	            #iqUDT_ConveyorInterface.VFDatSpeed := #sx_SpeedSetpointReached AND
	            #sx_AixAvailableControler AND
	            #si_ActualSpeed <> 0 AND
	            NOT #sx_SpeedFeedbackError;             // Copy setpoint speed reached state from static to the output conveyor interface structure

	            #iqUDT_ConveyorInterface.InternalWarningVFD := #sUDT_HMIStatus.PNSlaveWarning;                                                       // Set the internal warning bit if any warning is active

	            #iqUDT_ConveyorInterface.InternalErrorVFD := #sx_ErrorCMotor;                   // Set the internal error bit if any fault is active

	            #iqUDT_ConveyorInterface.ActualSpeed := ABS(#si_ActualSpeed);                   // Copy the calculated value to the output

	            #iqUDT_ConveyorInterface.ConfigurationError := #sx_ConfigurationError;          // Copy the calculated value to the output

	        END_IF;


	    END_REGION

	    REGION 10.2 - Move error status TO HMI Status

	        // Copy error status to output
	        #qUDT_HMIStatus := #sUDT_HMIStatus;

	    END_REGION

	END_REGION

	REGION 11 - Statistic

	    REGION 11.1 - General
	        // Statement section REGION
	        #sx_GeneralStatisticsReset := #iqUDT_ConveyorInterface.ResetStatistics;
	    END_REGION

	    // Create trigger on error and create statistics for profinet slave not online
	    #sR_TRIG_PNSlaveNotOnline(CLK := #sUDT_HMIStatus.PNSlaveNotOnline);                 // Detect the rising edge of the error

	    IF #sx_GeneralStatisticsReset OR #sUDT_HMIStatus.PNSlaveNotOnline
	    THEN

	        "FC_Statistics"(ix_Reset := #sx_GeneralStatisticsReset,
	                        ix_Activate := #sUDT_HMIStatus.PNSlaveNotOnline,
	                        ix_RTrigActivate := #sR_TRIG_PNSlaveNotOnline.Q,
	                        iqUDT_Statistics := #iqUDT_MCOStatistics.PNSlaveNotOnline);

	        #iqUDT_MCOStatistics.PNSlaveNotOnline := #iqUDT_MCOStatistics.PNSlaveNotOnline;
	    END_IF;

	    // Create trigger on error and create statistics for profinet slave error
	    #sR_TRIG_PNSlaveError(CLK := #sUDT_HMIStatus.PNSlaveError);                                                                          // Detect the rising edge of the error

	    IF #sx_GeneralStatisticsReset OR #sUDT_HMIStatus.PNSlaveError
	    THEN

	        "FC_Statistics"(ix_Reset := #sx_GeneralStatisticsReset,
	                        ix_Activate := #sUDT_HMIStatus.PNSlaveError,
	                        ix_RTrigActivate := #sR_TRIG_PNSlaveError.Q,
	                        iqUDT_Statistics := #iqUDT_MCOStatistics.PNSlaveError);

	        #iqUDT_MCOStatistics.PNSlaveError := #iqUDT_MCOStatistics.PNSlaveError;
	    END_IF;


	    // Create trigger on error and create statistics for MCO communication error
	    #sR_TRIG_CommunicationErrorMCO(CLK := #qUDT_HMIStatus.CommunicationErrorVFD);            // Detect the rising edge of the error

	    IF #sx_GeneralStatisticsReset OR #qUDT_HMIStatus.CommunicationErrorVFD
	    THEN

	        "FC_Statistics"(ix_Reset := #sx_GeneralStatisticsReset,
	                        ix_Activate := #qUDT_HMIStatus.CommunicationErrorVFD,
	                        ix_RTrigActivate := #sR_TRIG_CommunicationErrorMCO.Q,
	                        iqUDT_Statistics := #iqUDT_MCOStatistics.CommunicationErrorMovikit);

	    END_IF;

	    REGION 11.1 - Motor

	        // Create trigger on error and create statistics for internal MCO Error
	        #sR_TRIG_MCOInternalError(CLK := #sUDT_HMIStatus.InternalError);         // Detect the rising edge of the error

	        IF #iqUDT_ConveyorInterface.ResetStatistics OR #sUDT_HMIStatus.InternalError
	        THEN

	            "FC_Statistics"(ix_Reset := #iqUDT_ConveyorInterface.ResetStatistics,
	                            ix_Activate := #sUDT_HMIStatus.InternalError,
	                            ix_RTrigActivate := #sR_TRIG_MCOInternalError.Q,
	                            iqUDT_Statistics := #iqUDT_MCOStatistics.VFDInternalError);

	        END_IF;

	        // Create trigger on running signal and create statistics for running status
	        #sR_TRIG_Running(CLK := #iqUDT_ConveyorInterface.VFDRunning);                           // Detect the rising edge of the signal

	        IF #iqUDT_ConveyorInterface.ResetStatistics OR #iqUDT_ConveyorInterface.VFDRunning
	        THEN

	            "FC_Statistics"(ix_Reset := #iqUDT_ConveyorInterface.ResetStatistics,
	                            ix_Activate := #iqUDT_ConveyorInterface.VFDRunning,
	                            ix_RTrigActivate := #sR_TRIG_Running.Q,
	                            iqUDT_Statistics := #iqUDT_MCOStatistics.Running);
	        END_IF;


	    END_REGION
	    REGION 12 Status bit allocation
	        "FC_BitAllocation"(ix_Bit0 := #qUDT_HMIStatus.SpeedFeedbackError,
	                           ix_Bit1 := #qUDT_HMIStatus.InternalWarning,
	                           ix_Bit2 := #qUDT_HMIStatus.InternalError,
	                           ix_Bit3 := #qUDT_HMIStatus.CommunicationErrorVFD,
	                           ix_Bit4 := #qUDT_HMIStatus.PNSlaveNotOnline,
	                           ix_Bit5 := #qUDT_HMIStatus.PNSlaveError,
	                           ix_Bit6 := #qUDT_HMIStatus.PNSlaveWarning,
	                           ix_Bit7 := FALSE,
	                           ix_Bit8 := FALSE,
	                           ix_Bit9 := FALSE,
	                           ix_Bit10 := FALSE,
	                           ix_Bit11 := FALSE,
	                           ix_Bit12 := FALSE,
	                           ix_Bit13 := FALSE,
	                           ix_Bit14 := FALSE,
	                           ix_Bit15 := FALSE,
	                           ix_Bit16 := FALSE,
	                           ix_Bit17 := FALSE,
	                           ix_Bit18 := FALSE,
	                           ix_Bit19 := FALSE,
	                           ix_Bit20 := FALSE,
	                           ix_Bit21 := FALSE,
	                           ix_Bit22 := FALSE,
	                           ix_Bit23 := FALSE,
	                           ix_Bit24 := FALSE,
	                           ix_Bit25 := FALSE,
	                           ix_Bit26 := FALSE,
	                           ix_Bit27 := FALSE,
	                           ix_Bit28 := FALSE,
	                           ix_Bit29 := FALSE,
	                           ix_Bit30 := FALSE,
	                           ix_Bit31 := FALSE,
	                           qdw_Dword => #qUDT_HMIStatus.ControllerStatus);
	    END_REGION
	END_REGION
END_FUNCTION_BLOCK

FUNCTION_BLOCK "FB_GateSection"
{ S7_Optimized_Access := 'TRUE' }
VERSION : 0.1
// ATTRIBUTES
// AUTO_NUMBER = True
// BLOCK_NUMBER = 213
// END_ATTRIBUTES
   VAR_INPUT
      ix_GateOpen { ExternalAccessible := 'False'; ExternalVisible := 'False'; ExternalWritable := 'False'} : Bool;   // When TRUE gate is open, when FALSE gate is close
      ix_OperatorButton { ExternalAccessible := 'False'; ExternalVisible := 'False'; ExternalWritable := 'False'} : Bool;   // When TRUE then operator button is pressed
      iudi_TimeOnDelay { ExternalAccessible := 'False'; ExternalVisible := 'False'; ExternalWritable := 'False'} : UDInt;   // Time on delay to enable the horn when the gate is closed
   END_VAR

   VAR_OUTPUT
      qx_Horn { ExternalAccessible := 'False'; ExternalVisible := 'False'; ExternalWritable := 'False'} : Bool;   // When TRUE enable horn sound
      qUDT_HMIStatus { ExternalAccessible := 'False'; ExternalVisible := 'False'; ExternalWritable := 'False'} : "UDT_GateStatus";   // HMI status structure
   END_VAR

   VAR
      sFB_GateIsClosed { ExternalAccessible := 'False'; ExternalVisible := 'False'; ExternalWritable := 'False'; S7_SetPoint := 'False'} : "FB_TimerOnOffDelay";   // Timer on delay to enable the horn signal when the gate is closed
      sR_TRIG_OperatorButton {InstructionName := 'R_TRIG'; LibVersion := '1.0'; ExternalAccessible := 'False'; ExternalVisible := 'False'; ExternalWritable := 'False'; S7_SetPoint := 'False'} : R_TRIG;   // Rising edge trigger operator button
      sx_GateClosedAndNoOperatorPresent { ExternalAccessible := 'False'; ExternalVisible := 'False'; ExternalWritable := 'False'} : Bool;   // Auxiliary variable TRUE when the gare is closed and no operator is present
   END_VAR


BEGIN
	(*
	----------------------------------------------------------------------------------------

	Version history:
	Date        | Version   | Author        | Remark
	----------------------------------------------------------------------------------------
	26/01/2022  | 0.0       | M. Piela      | first release TIA 15.1
	21/02/2023  | 4.0       | F.Baten       | 4.0 Release TIA 17.5
	 *)

	REGION 1 - Push button trigger

	    #sR_TRIG_OperatorButton(CLK := #ix_OperatorButton);  //Operator button

	END_REGION

	REGION 2 - Gate open time counting

	    //Enable the horn signal when the gate is closed for 10 minutes
	    #sFB_GateIsClosed(iudi_OnDelayTime := #iudi_TimeOnDelay,
	                      ix_SignalToDelay := NOT #ix_GateOpen AND NOT #sR_TRIG_OperatorButton.Q,
	                      ix_Enable := TRUE,
	                      qx_DelayedSignal => #sx_GateClosedAndNoOperatorPresent);

	END_REGION

	REGION 3 - Status

	    #qUDT_HMIStatus.Specific.GateClosed := NOT #ix_GateOpen;
	    #qUDT_HMIStatus.Specific.GateClosedAndNoOperatorPresent := #sx_GateClosedAndNoOperatorPresent;

	    IF NOT #qUDT_HMIStatus.Specific.GateClosed
	    THEN
	        #qUDT_HMIStatus.Status := "DB_HMIStatusConfiguration".GateOpen;
	    END_IF;

	    IF #qUDT_HMIStatus.Specific.GateClosed
	    THEN
	        #qUDT_HMIStatus.Status := "DB_HMIStatusConfiguration".GateClosed;
	    END_IF;

	    IF #qUDT_HMIStatus.Specific.GateClosedAndNoOperatorPresent
	    THEN
	        #qUDT_HMIStatus.Status := "DB_HMIStatusConfiguration".GateClosedAndNoOperatorPresent;
	    END_IF;


	END_REGION


	REGION 4 - Output enable

	    #qx_Horn := #sx_GateClosedAndNoOperatorPresent;

	END_REGION
END_FUNCTION_BLOCK

FUNCTION_BLOCK "FB_Inching"
{ S7_Optimized_Access := 'TRUE' }
VERSION : 0.1
// ATTRIBUTES
// AUTO_NUMBER = True
// BLOCK_NUMBER = 214
// END_ATTRIBUTES
   VAR_INPUT
      iUDT_InchingConfiguration { ExternalAccessible := 'False'; ExternalVisible := 'False'; ExternalWritable := 'False'} : "UDT_InchingConfiguration";   //  Inching configuration structure
      iUDT_FeedConveyorConfiguration { ExternalAccessible := 'False'; ExternalVisible := 'False'; ExternalWritable := 'False'} : "UDT_ConveyorConfiguration";   //  Feed conveyor configuration structure
      iUDT_ConveyorConfiguration { ExternalAccessible := 'False'; ExternalVisible := 'False'; ExternalWritable := 'False'} : "UDT_ConveyorConfiguration";   //  Conveyor configuration structure
      ii_PECEoSDistanceUpstream { ExternalAccessible := 'False'; ExternalVisible := 'False'; ExternalWritable := 'False'} : DInt;   //  Distance between photo eye and the end of conveyor [mm]
      ii_PECEoSDistance { ExternalAccessible := 'False'; ExternalVisible := 'False'; ExternalWritable := 'False'} : DInt;   //  Distance between photo eye and the end of conveyor [mm]
      ix_PECEoS { ExternalAccessible := 'False'; ExternalVisible := 'False'; ExternalWritable := 'False'} : Bool;   //  PEC signal End of Section
      ix_Release { ExternalAccessible := 'False'; ExternalVisible := 'False'; ExternalWritable := 'False'} : Bool;   //  Release button
      ix_Clockpulse1 { ExternalAccessible := 'False'; ExternalVisible := 'False'; ExternalWritable := 'False'} : Bool;   //  Clock pulse to flash when emptying
      ix_Clockpulse2 { ExternalAccessible := 'False'; ExternalVisible := 'False'; ExternalWritable := 'False'} : Bool;   //  Clock pulse to flash when emptied
   END_VAR

   VAR_OUTPUT
      qx_ExternalRequestHold { ExternalAccessible := 'False'; ExternalVisible := 'False'; ExternalWritable := 'False'} : Bool;   //  External output to request conveyor hold
      qx_ExternalRequestDieBack { ExternalAccessible := 'False'; ExternalVisible := 'False'; ExternalWritable := 'False'} : Bool;   //  External output to request die back
      qx_IndicationSignal { ExternalAccessible := 'False'; ExternalVisible := 'False'; ExternalWritable := 'False'} : Bool;   //  Output to indication: flashing with clockpuls 1 then emptying, flashing with clockpuls 2 then emptied, continuously on then full
   END_VAR

   VAR_IN_OUT
      iqUDT_FeedConveyor : "UDT_ConveyorInterface";   //  Feed conveyor interface structure
      iqUDT_InchingConveyor : "UDT_ConveyorInterface";   //  Inching conveyor interface structure
      iqUDT_HandShakeUp : "UDT_ConveyorHandshake";   //  Conveyor handshake structure
   END_VAR

   VAR
      sFB_ButtonTimerFull { ExternalAccessible := 'False'; ExternalVisible := 'False'; ExternalWritable := 'False'; S7_SetPoint := 'False'} : "FB_TimerOnOffDelay";   //  Delaytime of the release button to set the conveyor full
      sFB_ButtonTimerRelease { ExternalAccessible := 'False'; ExternalVisible := 'False'; ExternalWritable := 'False'; S7_SetPoint := 'False'} : "FB_TimerOnOffDelay";   //  Delaytime of the release button to release the conveyor to emty
      sR_TRIG_RTSUp {InstructionName := 'R_TRIG'; LibVersion := '1.0'; ExternalAccessible := 'False'; ExternalVisible := 'False'; ExternalWritable := 'False'; S7_SetPoint := 'False'} : R_TRIG;   //  Rising edge trigger ready to send upstream
      sR_TRIG_TIP {InstructionName := 'R_TRIG'; LibVersion := '1.0'; ExternalAccessible := 'False'; ExternalVisible := 'False'; ExternalWritable := 'False'; S7_SetPoint := 'False'} : R_TRIG;   //  Rising edge trigger tip
      sF_TRIG_PECEoS {InstructionName := 'F_TRIG'; LibVersion := '1.0'; ExternalAccessible := 'False'; ExternalVisible := 'False'; ExternalWritable := 'False'; S7_SetPoint := 'False'} : F_TRIG;   //  Falling edge trigger PEC EoS
      sdi_FirstParcelPosition { ExternalAccessible := 'False'; ExternalVisible := 'False'; ExternalWritable := 'False'} : DInt;   //  The position the front of the first parcel is where '0' is end of conveyor [cm]
      sdi_ActualGapCounter { ExternalAccessible := 'False'; ExternalVisible := 'False'; ExternalWritable := 'False'} : DInt;   //  The number of centimeters the conveyor has to run to complete the gap
      sdi_ActualRunningEmpty { ExternalAccessible := 'False'; ExternalVisible := 'False'; ExternalWritable := 'False'} : DInt;   //  The number of centimeters the conveyor has to run to run empty
      sdi_ActualTIPDistance { ExternalAccessible := 'False'; ExternalVisible := 'False'; ExternalWritable := 'False'} : DInt;   //  Actual distance befor TIP will be activated
      sdi_FullDegree { ExternalAccessible := 'False'; ExternalVisible := 'False'; ExternalWritable := 'False'} : DInt;   //  Filling degree
      sx_Emptied { ExternalAccessible := 'False'; ExternalVisible := 'False'; ExternalWritable := 'False'} : Bool;   //  Inching conveyor condition is emptied, wait to start
      sx_Inching { ExternalAccessible := 'False'; ExternalVisible := 'False'; ExternalWritable := 'False'} : Bool;   //  Inching conveyor condition is inching
      sx_Full { ExternalAccessible := 'False'; ExternalVisible := 'False'; ExternalWritable := 'False'} : Bool;   //  Inching conveyor condition is full
      sx_Emptying { ExternalAccessible := 'False'; ExternalVisible := 'False'; ExternalWritable := 'False'} : Bool;   //  Inching conveyor condition is emptying
      sx_Run { ExternalAccessible := 'False'; ExternalVisible := 'False'; ExternalWritable := 'False'} : Bool;   //  Run inching conveyor (release hold)
      sx_FirstParcel { ExternalAccessible := 'False'; ExternalVisible := 'False'; ExternalWritable := 'False'} : Bool;   //  First parcel entering the inching conveyor
      sx_UpdateFirst { ExternalAccessible := 'False'; ExternalVisible := 'False'; ExternalWritable := 'False'} : Bool;   //  The first parcel has entered the PEC
      sx_ReleaseButton { ExternalAccessible := 'False'; ExternalVisible := 'False'; ExternalWritable := 'False'} : Bool;   //  Release button is pressed to set Full condidition, first release the button to set Release function
   END_VAR

   VAR CONSTANT
      ci_Startvalue : Int := 2;
   END_VAR


BEGIN
	(*
	----------------------------------------------------------------------------------------

	Version history:
	Date        | Version   | Author        | Remark
	----------------------------------------------------------------------------------------
	28/10/2019  | 3.0       | F.Baten       | first release TIA 15
	14/01/2020  | 3.1       | F.Baten       | Updatet "UDT_ConveyorConfiguration"
	22/04/2020  | 3.2       | L.Klar        | Adjusted after conveyor UDT's change
	21/02/2023  | 4.0       | F.Baten       | 4.0 Release TIA 17.5
	*)

	REGION 1 - Triggers

	    // Beginning of transporting the parcel in.
	    #sR_TRIG_TIP(CLK := #iqUDT_HandShakeUp.TIP);

	    // The upstream conveyor is ready to transport.
	    #sR_TRIG_RTSUp(CLK := #iqUDT_HandShakeUp.RTS);

	    // Falling edge trigger PEC EoS.
	    #sF_TRIG_PECEoS(CLK := #ix_PECEoS);

	END_REGION

	REGION 2 - Set distances

	    REGION 2.1 - Set the desired gap distance when the TIP starts.

	        // The actual starting of the inching conveyor is the offset earlier so that has to be deducted from the desired gap.
	        IF #sR_TRIG_TIP.Q
	        THEN
	            // Distance the parcel starts at the tipping position is smaller than the disired gapsize.
	            IF (#iUDT_FeedConveyorConfiguration.Forward_Direction.PEC_EoSDistanceOffset / 10) < #iUDT_InchingConfiguration.GapSize
	            THEN
	                // Then decrease the gapsize (to be done at the inching conveyor) with the offset because both conveyors are running when the TIP is active.
	                #sdi_ActualGapCounter :=
	                #iUDT_InchingConfiguration.GapSize -
	                (#iUDT_FeedConveyorConfiguration.Forward_Direction.PEC_EoSDistanceOffset / 10) -
	                #ci_Startvalue;
	            ELSE
	                // The distance for the gap is already covered by the offset distance.
	                #sdi_ActualGapCounter := 0;
	            END_IF;
	        END_IF;

	    END_REGION

	    REGION 2.2 - Track the parcel on the upstream conveyor

	        //  Set the distance from the trigger signal until the point the TIP would start.
	        IF #sR_TRIG_RTSUp.Q
	        THEN
	            // PEC distance - Offset = TIP distance on the upstream conveyor.
	            #sdi_ActualTIPDistance := (#ii_PECEoSDistanceUpstream - #iUDT_FeedConveyorConfiguration.Forward_Direction.PEC_EoSDistanceOffset) / 10;
	            IF #sdi_ActualTIPDistance < 0
	            THEN
	                #sdi_ActualTIPDistance := 0;
	            END_IF;
	        END_IF;

	    END_REGION

	    REGION 2.3 - Update the first parcel position

	        IF #sF_TRIG_PECEoS.Q
	            AND NOT #sx_UpdateFirst
	        THEN
	            // Set the position of the PEC as the first parcel position.
	            #sdi_FirstParcelPosition := #ii_PECEoSDistance / 10;
	            // First parcel is updated.
	            #sx_UpdateFirst := TRUE;
	        END_IF;

	    END_REGION

	END_REGION

	REGION 3 - Button

	    // When the button is pressed for a longer time it is accepted as setting full action.
	    #sFB_ButtonTimerRelease(iudi_OnDelayTime := #iUDT_InchingConfiguration.ButtonReleaseDelayTime,
	                            iudi_OffDelayTime := 0,
	                            ix_SignalToDelay := #sx_Full AND #ix_Release AND NOT #sx_ReleaseButton);

	    // When the button is pressed for a longer time it is accepted as release action.
	    #sFB_ButtonTimerFull(iudi_OnDelayTime := #iUDT_InchingConfiguration.ButtonReleaseDelayTime,
	                         iudi_OffDelayTime := 0,
	                         ix_SignalToDelay := #sx_Inching AND #ix_Release);

	    #sx_ReleaseButton := (#sx_Inching
	    OR #sx_ReleaseButton)
	    AND #ix_Release;

	    // When full, the release is started by the release button.
	    IF #sx_Full
	        AND #sFB_ButtonTimerRelease.qx_DelayedSignal
	    THEN
	        #sx_Emptying := TRUE;
	    END_IF;

	END_REGION

	REGION 4 - Displacement update

	    REGION 4.1 - Update the gap between the parcel and the beginning of the conveyor

	        // The Inching conveyor is allowed to run and not transferring to upstream and the gapcounter is still bigger than '0'.
	        IF #sx_Run
	            AND NOT #iqUDT_HandShakeUp.TIP
	            AND #sdi_ActualGapCounter > 0
	        THEN
	            // Decrease the counter by the conveyors displacement.
	            #sdi_ActualGapCounter -= #iqUDT_InchingConveyor.Displacement;
	            IF #sdi_ActualGapCounter < 0
	            THEN
	                #sdi_ActualGapCounter := 0;
	            END_IF;
	        END_IF;

	    END_REGION

	    REGION 4.2 - Update the first parcel position (the head OF the cue)

	        // The counter is still bigger than '0'.
	        IF #sdi_FirstParcelPosition > 0
	        THEN
	            // Decrease the counter by the conveyors displacement.
	            #sdi_FirstParcelPosition -= #iqUDT_InchingConveyor.Displacement;
	            IF #sdi_FirstParcelPosition < 0
	            THEN
	                #sdi_FirstParcelPosition := 0;
	            END_IF;
	        END_IF;

	    END_REGION

	    REGION 4.3 - Update running empty distance

	        // The counter is still bigger than '0'.
	        IF #sdi_ActualRunningEmpty > 0
	            AND #sx_Emptying
	        THEN
	            // Decrease the counter by the conveyors displacement.
	            #sdi_ActualRunningEmpty -= #iqUDT_InchingConveyor.Displacement;
	            IF #sdi_ActualRunningEmpty < 0
	            THEN
	                #sdi_ActualRunningEmpty := 0;
	            END_IF;
	        END_IF;

	    END_REGION

	    REGION 4.4 - Update the parcel position on the upstream conveyor

	        // The counter is still bigger than '0'.
	        IF #sdi_ActualTIPDistance > 0
	        THEN
	            // Decrease the counter by the conveyors displacement.
	            #sdi_ActualTIPDistance -= #iqUDT_FeedConveyor.Displacement;
	            IF #sdi_ActualTIPDistance < 0
	            THEN
	                #sdi_ActualTIPDistance := 0;
	            END_IF;
	        END_IF;

	    END_REGION

	END_REGION


	REGION 5 - Status mode

	    (* The positions are counting back from the maximal to '0'.
	     When the inching conveyor is full, set the running empty distance. *)
	    IF (#sdi_FirstParcelPosition < #iUDT_InchingConfiguration.MaximalFillingPosition
	        AND #sx_FirstParcel
	        AND NOT #iqUDT_HandShakeUp.TIP
	        AND NOT #sx_Full)
	        OR (#sdi_FirstParcelPosition < 2
	        AND #sx_FirstParcel
	        AND NOT #sx_Full)
	        OR #sFB_ButtonTimerFull.qx_DelayedSignal
	    THEN
	        // The length of the conveyor is the run empty length.
	        #sdi_ActualRunningEmpty := #iUDT_ConveyorConfiguration.Common.Length / 10;
	        #sx_Full := TRUE;
	        #sx_Inching := FALSE;
	    END_IF;

	    // Running epmty and the distance is done.
	    IF #sx_Emptying
	        AND #sdi_ActualRunningEmpty <= 0
	    THEN
	        #sx_UpdateFirst := FALSE;
	        #sx_FirstParcel := FALSE;
	        #sx_Emptying := FALSE;
	        #sx_Full := FALSE;
	        #sx_Emptied := TRUE;
	    END_IF;

	    // Acknowledge from operator to start again.
	    IF #sx_Emptied
	        AND (#ix_Release
	        OR NOT #iUDT_InchingConfiguration.WaitForStartConf)
	    THEN
	        #sx_Inching := TRUE;
	        #sx_Emptied := FALSE;
	    END_IF;

	    // Activate first parcel.
	    IF #sx_Inching
	        AND NOT #sx_FirstParcel
	        AND #iqUDT_HandShakeUp.TIP
	    THEN
	        // Set the position the parcel actual is.
	        #sdi_FirstParcelPosition := (#iUDT_ConveyorConfiguration.Common.Length + #iUDT_FeedConveyorConfiguration.Forward_Direction.PEC_EoSDistanceOffset) / 10;
	        // Indicating the first parcel is detected.
	        #sx_FirstParcel := TRUE;
	    END_IF;

	    // If no mode is active the conveyor is set to full so an operator has to check and release.
	    IF NOT #sx_Emptied AND NOT #sx_Emptying AND NOT #sx_Full AND NOT #sx_Inching
	    THEN
	        #sx_Full := TRUE;
	    END_IF;

	END_REGION

	REGION 6 - Hold inching conveyor

	    (* Run inching conveyor
	       - inching mode - RTS signal and parcel is 1 cm before it will stop
	                      - Gap is not there yet
	       - running empty *)
	    #sx_Run :=
	    #sx_Inching
	    AND (((#iqUDT_HandShakeUp.RTS OR #iqUDT_HandShakeUp.TIP)
	    AND (#sdi_ActualTIPDistance < #ci_Startvalue)
	    OR #iqUDT_HandShakeUp.RTS
	    AND NOT (#iqUDT_FeedConveyor.RunFwd OR #iqUDT_FeedConveyor.RunRvs))
	    OR #sdi_ActualGapCounter > 1)
	    OR #sx_Emptying;

	    #qx_ExternalRequestHold := NOT #sx_Run;

	END_REGION

	REGION 7 - External dieback signal

	    (* Stop feeding in new parcels
	       - Gap has to be there
	       - Conveyor is full
	       - Conveyor is running empty *)
	    #qx_ExternalRequestDieBack :=
	    (#iqUDT_HandShakeUp.RTS
	    AND (#sdi_ActualGapCounter > 1)
	    AND NOT #iqUDT_HandShakeUp.TIP)
	    OR #sx_Full
	    OR #sx_Emptying;

	END_REGION

	REGION 8 - Signal

	    // Signalling full and emptying.
	    #qx_IndicationSignal :=
	    (NOT #sx_Emptying
	    AND #sx_Full)
	    OR (#sx_Emptying
	    AND #ix_Clockpulse1)
	    OR (#sx_Emptied
	    AND #ix_Clockpulse2);

	    // Percentage of conveyor used.
	    #sdi_FullDegree := 100 - (#sdi_FirstParcelPosition / (#iUDT_ConveyorConfiguration.Common.Length / 1000));

	END_REGION

END_FUNCTION_BLOCK

FUNCTION_BLOCK "FB_RIOVSU"
TITLE = FB_RIOVSU
{ S7_Optimized_Access := 'TRUE' }
AUTHOR : MHSE
FAMILY : GeneralSystemFunctions
VERSION : 3.0
// ATTRIBUTES
// AUTO_NUMBER = True
// BLOCK_NUMBER = 226
// END_ATTRIBUTES
   VAR_INPUT
      is_ET200spPNDeviceName { ExternalAccessible := 'False'; ExternalVisible := 'False'; ExternalWritable := 'False'} : String;   //   Name of the ET200sp device
      ix_400VintOk { ExternalAccessible := 'False'; ExternalVisible := 'False'; ExternalWritable := 'False'} : Bool;   //   TRUE if internal circuit breaker 400V is ok
      ix_400VextOk { ExternalAccessible := 'False'; ExternalVisible := 'False'; ExternalWritable := 'False'} : Bool;   //   TRUE if external 400V Main cabinet is ok
      ix_BrakeSupplyOk { ExternalAccessible := 'False'; ExternalVisible := 'False'; ExternalWritable := 'False'} : Bool;   //   TRUE if circuit breaker of brake power supply is ok
      ix_ThermalBrake { ExternalAccessible := 'False'; ExternalVisible := 'False'; ExternalWritable := 'False'} : Bool;   //   TRUE when No thermal error
      ix_24VOk { ExternalAccessible := 'False'; ExternalVisible := 'False'; ExternalWritable := 'False'} : Bool;   //   TRUE when 24V power supply to RIO is ok
      ix_SimulationModeActive { ExternalAccessible := 'False'; ExternalVisible := 'False'; ExternalWritable := 'False'} : Bool;   //   True when Simulation mode active
      ix_HardwareOk { ExternalAccessible := 'False'; ExternalVisible := 'False'; ExternalWritable := 'False'} : Bool;   //  TRUE when  hardware is Ok
   END_VAR

   VAR_OUTPUT
      qUDT_HMIStatus { ExternalAccessible := 'False'; ExternalVisible := 'False'; ExternalWritable := 'False'} : "UDT_RIOVSUStatus";   //   HMI status structure
   END_VAR

   VAR_IN_OUT
      iqUDT_Statistics : "UDT_RIOVSUStatistics";   //   Statistics structure
      iqUDT_VSUInterface : "UDT_VSUInterface";   //   Interface RIO and VSU
   END_VAR

   VAR
      sUDT_HMIStatus { ExternalAccessible := 'False'; ExternalVisible := 'False'; ExternalWritable := 'False'; S7_SetPoint := 'False'} : "UDT_RIOVSUStatus";   //   HMI status structure
      sUDT_PNDevice { ExternalAccessible := 'False'; ExternalVisible := 'False'; ExternalWritable := 'False'; S7_SetPoint := 'False'} : "UDT_PNDevice";   //   PN device structure
      sa_PNPortsStatus { ExternalAccessible := 'False'; ExternalVisible := 'False'; ExternalWritable := 'False'} : Array[1..8] of Bool;   // TRUE when specific port has an error
      sFB_TimerOnOffDelayCheckSupply { ExternalAccessible := 'False'; ExternalVisible := 'False'; ExternalWritable := 'False'; S7_SetPoint := 'False'} : "FB_TimerOnOffDelay";   //   MHS "TimerOnOffDelay" - to delay time for VFD supply contactor
      sR_TRIG_Int400VCBError {InstructionName := 'R_TRIG'; LibVersion := '1.0'; ExternalAccessible := 'False'; ExternalVisible := 'False'; ExternalWritable := 'False'; S7_SetPoint := 'False'} : R_TRIG;   //   Rising edge for trigger 400v internal error
      sR_TRIG_Int24VError {InstructionName := 'R_TRIG'; LibVersion := '1.0'; ExternalAccessible := 'False'; ExternalVisible := 'False'; ExternalWritable := 'False'; S7_SetPoint := 'False'} : R_TRIG;   //   Rising edge for trigger 24v internal error
      sR_TRIG_BrakeCBerror {InstructionName := 'R_TRIG'; LibVersion := '1.0'; ExternalAccessible := 'False'; ExternalVisible := 'False'; ExternalWritable := 'False'; S7_SetPoint := 'False'} : R_TRIG;   //   Rising edge for trigger brake circuit breaker tripped
      sR_TRIG_BrakeThermError {InstructionName := 'R_TRIG'; LibVersion := '1.0'; ExternalAccessible := 'False'; ExternalVisible := 'False'; ExternalWritable := 'False'; S7_SetPoint := 'False'} : R_TRIG;   //   Rising edge for trigger brake thermal error
      sR_TRIG_DeviceFound {InstructionName := 'R_TRIG'; LibVersion := '1.0'; ExternalAccessible := 'False'; ExternalVisible := 'False'; ExternalWritable := 'False'; S7_SetPoint := 'False'} : R_TRIG;   //   Rising edge for trigger scan modules
      sR_TRIG_PNSlaveNotOnline {InstructionName := 'R_TRIG'; LibVersion := '1.0'; ExternalAccessible := 'False'; ExternalVisible := 'False'; ExternalWritable := 'False'; S7_SetPoint := 'False'} : R_TRIG;   //   Rising edge for trigger Profinet slave not online statistics
      sR_TRIG_PNSlaveError {InstructionName := 'R_TRIG'; LibVersion := '1.0'; ExternalAccessible := 'False'; ExternalVisible := 'False'; ExternalWritable := 'False'; S7_SetPoint := 'False'} : R_TRIG;   //   Rising edge for trigger Profinet slave error statistics
      si_ModuleStateReturn { ExternalAccessible := 'False'; ExternalVisible := 'False'; ExternalWritable := 'False'} : Int;   //   Status structure
      si_NrOfModulesWithError { ExternalAccessible := 'False'; ExternalVisible := 'False'; ExternalWritable := 'False'} : Int;   //   Number of the faulty modules
      sx_PNSlaveOnline { ExternalAccessible := 'False'; ExternalVisible := 'False'; ExternalWritable := 'False'} : Bool;   //   Profinet device is online and error free
      sx_PowerOk { ExternalAccessible := 'False'; ExternalVisible := 'False'; ExternalWritable := 'False'} : Bool;   //   True = External Power OK
      sx_ConfigurationError { ExternalAccessible := 'False'; ExternalVisible := 'False'; ExternalWritable := 'False'} : Bool;   //   Commissioning: configuration error
   END_VAR

   VAR_TEMP
      ta_Configured : Array[0..127] of Bool;   //   Configured modules array
      ta_Exist : Array[0..127] of Bool;   //   Existing modules array
      ta_Error : Array[0..127] of Bool;   //   Faulty modules array
      ti_NrOfModule : Int;   //   Number of current module
      ti_DiagArraySize : Int;   //   Diagnostic array size
   END_VAR

   VAR CONSTANT
      cui_ConfiguredModulesMode : UInt := 1;   //   Mode selector: 1 = Configured modules scan mode
      cui_ModuleErrorMode : UInt := 2;   //   Mode selector: 2 = Existing modules scan mode
      cui_ExistingModulesMode : UInt := 4;   //   Mode selector: 3 = Module Error scan mode
      ci_PowerSupplyDelayTime : UInt := 4000;   //   Power supply delay time
      ci_NumberOfProfinetPorts : Int := 2;   // Number of Profinet ports in device
   END_VAR


BEGIN
	(*
	----------------------------------------------------------------------------------------

	Version history:
	Date        | Version   | Author        | Remark
	----------------------------------------------------------------------------------------
	03/09-2019  | 2.1       | F.Baten       | first release MHS TIA 15.1
	23/09/2019  | 2.2       | F.Baten       | Changed region 1 contents to FC
	12/10/2019  | 2.3       | L. Klar       | Updated status structure
	14/10/2019  | 2.4       | S. Deulkar    | Added equipment control structure and created
	                                        | region for status
	12/11/2019  | 3.0       | P.Majka       | 3.0 MHS library release TIA 15.1
	29/11/2019  | 3.1       | F.Baten       | Updated interface to VSU
	04/12/2019  | 3.2       | F.Baten       | Region 3: ix_SimulationModeActive rearranged to correct position
	09/12/2019  | 3.3       | F.Baten       | Region 5: added #ix_SimulationModeActive to PNDeviceOk
	04/03/2020  | 3.4       | F.Baten       | Updated errors and warnings and interface to VSU
	06/08/2020  | 3.5       | L.Klar        | Initialize the #si_NrOfModulesWithError on the reset
	03/11/2020  | 3.9       | K.Pokorski    | Profinet ports diagnostics added
	02/08/2021  | 3.5       | S. Deulkar    | Added logic to reset error when 24V is not okay.
	21/02/2023  | 4.0       | F.Baten       | 4.0 Release TIA 17.5
	*)

	REGION 1 - Get Device Profinet information

	    "FC_GetDevicePN"(is_PNDeviceName := #is_ET200spPNDeviceName,
	                     ix_SimulationModeActive := #ix_SimulationModeActive,
	                     iqUDT_PND := #sUDT_PNDevice);


	    "FC_GetPNPortStatus"(ii_NumberOfPorts := #ci_NumberOfProfinetPorts,
	                         iUDT_DevicePNInfo := #sUDT_PNDevice,
	                         qa_PortFault => #sa_PNPortsStatus);

	END_REGION

	REGION 2 - Reset errors
	    // reset Profinet Slave error/not online
	    IF #iqUDT_VSUInterface.InternalErrorReset
	        OR NOT #ix_24VOk
	    THEN
	        #sUDT_HMIStatus."400VCircuitBreaker" := FALSE;
	        #sUDT_HMIStatus.BrakeCircuitBreaker := FALSE;
	        #sUDT_HMIStatus.BrakeThermalError := FALSE;
	        #sUDT_HMIStatus.PNSlaveNotOnline := FALSE;
	        #sUDT_HMIStatus.PNSlaveError := FALSE;
	        #sUDT_HMIStatus."24VPowersupplyError" := FALSE;
	        #sUDT_HMIStatus.PNSlaveWarning := FALSE;
	        #si_NrOfModulesWithError := 0;

	    END_IF;

	    // reset ET200sp module error status
	    IF #sUDT_HMIStatus.PNSlaveNotOnline OR #iqUDT_VSUInterface.InternalErrorReset OR NOT #ix_24VOk
	    THEN
	        FILL_BLK(IN := FALSE,
	                 COUNT := 32,
	                 OUT => #sUDT_HMIStatus.ET200sp_ErrorModule[0]);
	    END_IF;

	END_REGION

	REGION 3 - Update PN slave device status
	    // Hardware will only be available after the delay, so the device has time for the initialisation
	    #sFB_TimerOnOffDelayCheckSupply(iudi_OnDelayTime := #ci_PowerSupplyDelayTime,
	                                    ix_SignalToDelay := #ix_24VOk,
	                                    qx_DelayedSignal => #sx_PowerOk);

	    // check if PN device is online
	    IF ((NOT "DB_ProfinetDiagnostic".ProfinetNetworks[#sUDT_PNDevice.PNNetworknumber].DeviceStatus[#sUDT_PNDevice.PNDeviceNumber].DeviceState.Exist
	        AND #sx_PowerOk)
	        OR NOT #sUDT_PNDevice.PNDeviceFound)
	        AND NOT #ix_SimulationModeActive
	    THEN
	        #sUDT_HMIStatus.PNSlaveNotOnline := TRUE;
	    END_IF;

	    // Check if PN ports are healthy
	    IF #sa_PNPortsStatus[1] XOR #sa_PNPortsStatus[2] THEN
	        #sUDT_HMIStatus.PNSlaveWarning := TRUE;
	    END_IF;

	    // check if PN device has an error
	    IF "DB_ProfinetDiagnostic".ProfinetNetworks[#sUDT_PNDevice.PNNetworknumber].DeviceStatus[#sUDT_PNDevice.PNDeviceNumber].DeviceState.Error
	        AND #sx_PowerOk
	        AND NOT #ix_SimulationModeActive
	        AND NOT #sUDT_HMIStatus.PNSlaveWarning

	    THEN
	        #sUDT_HMIStatus.PNSlaveError := TRUE;
	    END_IF;

	    // set bit when PN device is healthy (online and no error)
	    #sx_PNSlaveOnline := NOT #sUDT_HMIStatus.PNSlaveNotOnline
	    AND #sUDT_PNDevice.PNDeviceFound
	    AND #sx_PowerOk
	    OR #ix_SimulationModeActive;

	    // create rising edge to scan module status when device is found
	    #sR_TRIG_DeviceFound(CLK := #sUDT_PNDevice.PNDeviceFound);

	END_REGION

	REGION 4 - Status update modules ET200sp
	    // update ET200sp module status
	    IF (#sx_PNSlaveOnline
	        AND (#sUDT_HMIStatus.PNSlaveError
	        OR #sUDT_HMIStatus.PNSlaveWarning))
	        OR #sR_TRIG_DeviceFound.Q
	    THEN
	        // get configured modules
	        #si_ModuleStateReturn := ModuleStates(LADDR := "DB_ProfinetDiagnostic".ProfinetNetworks[#sUDT_PNDevice.PNNetworknumber].DeviceStatus[#sUDT_PNDevice.PNDeviceNumber].DeviceState.HW_ID,
	                                              MODE := #cui_ConfiguredModulesMode,
	                                              STATE := #ta_Configured);

	        // get module online status
	        #si_ModuleStateReturn := ModuleStates(LADDR := "DB_ProfinetDiagnostic".ProfinetNetworks[#sUDT_PNDevice.PNNetworknumber].DeviceStatus[#sUDT_PNDevice.PNDeviceNumber].DeviceState.HW_ID,
	                                              MODE := #cui_ExistingModulesMode,
	                                              STATE := #ta_Exist);

	        // get module error status
	        #si_ModuleStateReturn := ModuleStates(LADDR := "DB_ProfinetDiagnostic".ProfinetNetworks[#sUDT_PNDevice.PNNetworknumber].DeviceStatus[#sUDT_PNDevice.PNDeviceNumber].DeviceState.HW_ID,
	                                              MODE := #cui_ModuleErrorMode,
	                                              STATE := #ta_Error);

	        // Handle ET200sp module errors/offline
	        IF (#si_ModuleStateReturn = 0)
	        THEN
	            #si_NrOfModulesWithError := 0;

	            #ti_DiagArraySize := "FC_GetNrOfArrayEl"(iv_Array := "DB_ProfinetDiagnostic".ProfinetNetworks[#sUDT_PNDevice.PNNetworknumber].DeviceStatus[#sUDT_PNDevice.PNDeviceNumber].Module);

	            FOR #ti_NrOfModule := 0 TO (#ti_DiagArraySize - 1) DO

	                // check if the module is configured
	                IF (#ta_Configured[#ti_NrOfModule])
	                THEN
	                    "DB_ProfinetDiagnostic".ProfinetNetworks[#sUDT_PNDevice.PNNetworknumber].DeviceStatus[#sUDT_PNDevice.PNDeviceNumber].Module[#ti_NrOfModule].Configured := TRUE;
	                    // and check if the module is online
	                    IF (#ta_Exist[#ti_NrOfModule])
	                    THEN
	                        "DB_ProfinetDiagnostic".ProfinetNetworks[#sUDT_PNDevice.PNNetworknumber].DeviceStatus[#sUDT_PNDevice.PNDeviceNumber].Module[#ti_NrOfModule].Exist := TRUE;

	                    ELSE
	                        "DB_ProfinetDiagnostic".ProfinetNetworks[#sUDT_PNDevice.PNNetworknumber].DeviceStatus[#sUDT_PNDevice.PNDeviceNumber].Module[#ti_NrOfModule].Exist := FALSE;
	                        #sUDT_HMIStatus.ET200sp_ErrorModule[#ti_NrOfModule] := TRUE;
	                        // count number of modules with error/offline
	                        #si_NrOfModulesWithError += 1;
	                    END_IF;

	                    // and check if the module has an error
	                    IF (NOT #ta_Error[#ti_NrOfModule])
	                    THEN
	                        "DB_ProfinetDiagnostic".ProfinetNetworks[#sUDT_PNDevice.PNNetworknumber].DeviceStatus[#sUDT_PNDevice.PNDeviceNumber].Module[#ti_NrOfModule].Error := FALSE;

	                    ELSE
	                        "DB_ProfinetDiagnostic".ProfinetNetworks[#sUDT_PNDevice.PNNetworknumber].DeviceStatus[#sUDT_PNDevice.PNDeviceNumber].Module[#ti_NrOfModule].Error := TRUE;
	                        #sUDT_HMIStatus.ET200sp_ErrorModule[#ti_NrOfModule] := TRUE;
	                        // count number OF modules with error/offline
	                        #si_NrOfModulesWithError += 1;
	                    END_IF;

	                ELSE
	                    // reset module status when module is not configured
	                    "DB_ProfinetDiagnostic".ProfinetNetworks[#sUDT_PNDevice.PNNetworknumber].DeviceStatus[#sUDT_PNDevice.PNDeviceNumber].Module[#ti_NrOfModule].Configured := FALSE;
	                    "DB_ProfinetDiagnostic".ProfinetNetworks[#sUDT_PNDevice.PNNetworknumber].DeviceStatus[#sUDT_PNDevice.PNDeviceNumber].Module[#ti_NrOfModule].Exist := FALSE;
	                    "DB_ProfinetDiagnostic".ProfinetNetworks[#sUDT_PNDevice.PNNetworknumber].DeviceStatus[#sUDT_PNDevice.PNDeviceNumber].Module[#ti_NrOfModule].Error := FALSE;

	                END_IF;
	            END_FOR;
	        END_IF;
	    END_IF;

	END_REGION

	REGION 5 - Check RIO Panel Status

	    // create 400v internal error
	    IF NOT #ix_400VintOk
	    THEN
	        #sUDT_HMIStatus."400VCircuitBreaker" := TRUE;
	    END_IF;

	    // create error circuit breaker brake tripped
	    IF NOT #ix_BrakeSupplyOk
	    THEN
	        #sUDT_HMIStatus.BrakeCircuitBreaker := TRUE;
	    END_IF;

	    // Create error thermal overload brake
	    IF NOT #ix_ThermalBrake
	    THEN
	        #sUDT_HMIStatus.BrakeThermalError := TRUE;
	    END_IF;

	    // Create error thermal overload brake
	    IF NOT #ix_24VOk
	    THEN
	        #sUDT_HMIStatus."24VPowersupplyError" := TRUE;
	    END_IF;

	    // check if 400 v to VFD positioning is ok
	    #iqUDT_VSUInterface.VSUMainPowerOk := #ix_400VextOk;

	    // set config not ok bit if no device found
	    #sx_ConfigurationError := NOT #sUDT_PNDevice.PNDeviceFound;

	END_REGION

	REGION 6 - Statistics
	    // create trigger on error and create statistics
	    #sR_TRIG_Int400VCBError(CLK := #sUDT_HMIStatus."400VCircuitBreaker");

	    IF #iqUDT_VSUInterface.ResetStatistics OR #sUDT_HMIStatus."400VCircuitBreaker"
	    THEN

	        "FC_Statistics"(ix_Reset := #iqUDT_VSUInterface.ResetStatistics,
	                        ix_Activate := #sUDT_HMIStatus."400VCircuitBreaker",
	                        ix_RTrigActivate := #sR_TRIG_Int400VCBError.Q,
	                        iqUDT_Statistics := #iqUDT_Statistics.Int400VCBError);
	    END_IF;

	    // create trigger on error and create statistics
	    #sR_TRIG_Int24VError(CLK := #sUDT_HMIStatus."24VPowersupplyError");

	    IF #iqUDT_VSUInterface.ResetStatistics OR #sUDT_HMIStatus."24VPowersupplyError"
	    THEN

	        "FC_Statistics"(ix_Reset := #iqUDT_VSUInterface.ResetStatistics,
	                        ix_Activate := #sUDT_HMIStatus."24VPowersupplyError",
	                        ix_RTrigActivate := #sR_TRIG_Int24VError.Q,
	                        iqUDT_Statistics := #iqUDT_Statistics."24VError");
	    END_IF;

	    // create trigger on error and create statistics
	    #sR_TRIG_BrakeCBerror(CLK := #sUDT_HMIStatus.BrakeCircuitBreaker);

	    IF #iqUDT_VSUInterface.ResetStatistics OR #sUDT_HMIStatus.BrakeCircuitBreaker
	    THEN

	        "FC_Statistics"(ix_Reset := #iqUDT_VSUInterface.ResetStatistics,
	                        ix_Activate := #sUDT_HMIStatus.BrakeCircuitBreaker,
	                        ix_RTrigActivate := #sR_TRIG_BrakeCBerror.Q,
	                        iqUDT_Statistics := #iqUDT_Statistics.BrakeCBerror);
	    END_IF;

	    // create trigger on error and create statistics
	    #sR_TRIG_BrakeThermError(CLK := #sUDT_HMIStatus.BrakeThermalError);

	    IF #iqUDT_VSUInterface.ResetStatistics OR #sUDT_HMIStatus.BrakeThermalError
	    THEN

	        "FC_Statistics"(ix_Reset := #iqUDT_VSUInterface.ResetStatistics,
	                        ix_Activate := #sUDT_HMIStatus.BrakeThermalError,
	                        ix_RTrigActivate := #sR_TRIG_BrakeThermError.Q,
	                        iqUDT_Statistics := #iqUDT_Statistics.BrakeThermError);
	    END_IF;

	    // create trigger on error and create statistics for profinet slave not online
	    #sR_TRIG_PNSlaveNotOnline(CLK := #sUDT_HMIStatus.PNSlaveNotOnline);

	    IF #iqUDT_VSUInterface.ResetStatistics OR #sUDT_HMIStatus.PNSlaveNotOnline
	    THEN

	        "FC_Statistics"(ix_Reset := #iqUDT_VSUInterface.ResetStatistics,
	                        ix_Activate := #sUDT_HMIStatus.PNSlaveNotOnline,
	                        ix_RTrigActivate := #sR_TRIG_PNSlaveNotOnline.Q,
	                        iqUDT_Statistics := #iqUDT_Statistics.PNSlaveNotOnline);
	    END_IF;

	    // create trigger on error and create statistics for profinet slave error
	    #sR_TRIG_PNSlaveError(CLK := #sUDT_HMIStatus.PNSlaveError);

	    IF #iqUDT_VSUInterface.ResetStatistics OR #sUDT_HMIStatus.PNSlaveError
	    THEN

	        "FC_Statistics"(ix_Reset := #iqUDT_VSUInterface.ResetStatistics,
	                        ix_Activate := #sUDT_HMIStatus.PNSlaveError,
	                        ix_RTrigActivate := #sR_TRIG_PNSlaveError.Q,
	                        iqUDT_Statistics := #iqUDT_Statistics.PNSlaveError);
	    END_IF;

	END_REGION

	REGION 7 - Status
	    // Statement section REGION
	    #iqUDT_VSUInterface.InternalErrorRIOPanel := #sUDT_HMIStatus.PNSlaveError
	    OR #sUDT_HMIStatus.PNSlaveNotOnline
	    OR #si_NrOfModulesWithError <> 0
	    OR #sUDT_HMIStatus."400VCircuitBreaker"
	    OR #sUDT_HMIStatus."24VPowersupplyError"
	    OR #sUDT_HMIStatus.BrakeCircuitBreaker
	    OR #sUDT_HMIStatus.BrakeThermalError;

	    // HMI status update

	    #qUDT_HMIStatus := #sUDT_HMIStatus;                       // Copy HMI status to output

	END_REGION

END_FUNCTION_BLOCK

FUNCTION_BLOCK "FB_XrayHS10080XCT"
TITLE = FB_Xray_HS10080XCT
{ S7_Optimized_Access := 'TRUE' }
AUTHOR : MHSE
FAMILY : Equipment
VERSION : 3.0
// ATTRIBUTES
// AUTO_NUMBER = True
// BLOCK_NUMBER = 44
// END_ATTRIBUTES
//Function block to control X-Ray.
   VAR_INPUT
      iUDT_EquipmentConfiguration { ExternalAccessible := 'False'; ExternalVisible := 'False'; ExternalWritable := 'False'} : "UDT_HS10080XCTConfiguration";   //  Configuration XCT 10080 structure
      iUDT_HMICommand { ExternalAccessible := 'False'; ExternalVisible := 'False'; ExternalWritable := 'False'} : "UDT_HS10080XCTHMICommand";   //  Command structure
      idi_TakeoutConveyorLength { ExternalAccessible := 'False'; ExternalVisible := 'False'; ExternalWritable := 'False'} : DInt;   //  Takeout Conveyor Length [mm]
      ix_SafetyReset { ExternalAccessible := 'False'; ExternalVisible := 'False'; ExternalWritable := 'False'} : Bool;   //  TRUE Safety reset command is active
      ix_SafetyOk { ExternalAccessible := 'False'; ExternalVisible := 'False'; ExternalWritable := 'False'} : Bool;   //  TRUE when Safety Circuit is healthy
      ix_24vOk { ExternalAccessible := 'False'; ExternalVisible := 'False'; ExternalWritable := 'False'} : Bool;   //  TRUE when 24VDC is healthy
      ix_400vOk { ExternalAccessible := 'False'; ExternalVisible := 'False'; ExternalWritable := 'False'} : Bool;   //  TRUE when 400VAC is healthy
      ix_ProfinetOk { ExternalAccessible := 'False'; ExternalVisible := 'False'; ExternalWritable := 'False'} : Bool;   //  TRUE when the PN node(s) of VSU are OK
      ix_Interlock { ExternalAccessible := 'False'; ExternalVisible := 'False'; ExternalWritable := 'False'} : Bool;   //  Contact from XCT . Closed: All doors are closed.Open: One of the doors of the tunnel is opened, machine is stopped
      ix_TempOutOfRange { ExternalAccessible := 'False'; ExternalVisible := 'False'; ExternalWritable := 'False'} : Bool;   //  Contact from XCT Closed: XCT doesn’t work because XCT operating temperature isn’t given. Open: XCT is in the right temperature range and it is possible to power on
      ix_PowerOn { ExternalAccessible := 'False'; ExternalVisible := 'False'; ExternalWritable := 'False'} : Bool;   //  The power-on acknowledgement. Open: The X-ray is shut down. Closed: The X-ray is turned on.
      ix_RepairSwitch { ExternalAccessible := 'False'; ExternalVisible := 'False'; ExternalWritable := 'False'} : Bool;   //  The main power switch. Open: Mains power on. Closed: Mains power off.
      ix_ServiceMode { ExternalAccessible := 'False'; ExternalVisible := 'False'; ExternalWritable := 'False'} : Bool;   //  Service mode state. Open: The X-ray is not in service mode. Closed: The X-ray is in service mode.
      ix_TransitActive { ExternalAccessible := 'False'; ExternalVisible := 'False'; ExternalWritable := 'False'} : Bool;   //  Transit mode state. Open: The transit mode is not active. Closed: The transit mode is active.
      ix_MachineOk { ExternalAccessible := 'False'; ExternalVisible := 'False'; ExternalWritable := 'False'} : Bool;   //  The X-ray is OK. Open: The X-ray has a fatal error; no operation is possible. Closed: The X-ray is initialised and working properly.
      ix_IQTestActive { ExternalAccessible := 'False'; ExternalVisible := 'False'; ExternalWritable := 'False'} : Bool;   //  TRUE when IQ test is active
      ix_CalReq { ExternalAccessible := 'False'; ExternalVisible := 'False'; ExternalWritable := 'False'} : Bool;   //  True when XCT is requesting callibration
      ix_AllowCalibration { ExternalAccessible := 'False'; ExternalVisible := 'False'; ExternalWritable := 'False'} : Bool;   //  Use to inhibit calibration in heavy flow if necessary
      ix_XrayReady { ExternalAccessible := 'False'; ExternalVisible := 'False'; ExternalWritable := 'False'} : Bool;   //  Ready to receive a bag state. Open: Not ready to receive a bag. Closed: X-ray is ready receive a bag.
      ix_PECInfeedEoS { ExternalAccessible := 'False'; ExternalVisible := 'False'; ExternalWritable := 'False'} : Bool;   //  TRUE when the end of section photoeye is not blocked
      ix_PECOutfeedEoS { ExternalAccessible := 'False'; ExternalVisible := 'False'; ExternalWritable := 'False'} : Bool;   //  TRUE when the end of section photoeye is not blocked
      ix_PECOutfeedPosition { ExternalAccessible := 'False'; ExternalVisible := 'False'; ExternalWritable := 'False'} : Bool;   //  TRUE when the data acailable at PEC position
      ix_InfConveyorError { ExternalAccessible := 'False'; ExternalVisible := 'False'; ExternalWritable := 'False'} : Bool;   //  Infeed conveyor error
      ix_MainSpeedOk { ExternalAccessible := 'False'; ExternalVisible := 'False'; ExternalWritable := 'False'} : Bool;   //  Main Conveyor speed OK. Open: The X-ray conveyor is not running or not running at specified speed. Closed: The X-ray conveyor is activated and running at specified speed.
      ix_OutfConveyorError { ExternalAccessible := 'False'; ExternalVisible := 'False'; ExternalWritable := 'False'} : Bool;   //  Outfeed Conveyor error.
      ix_NoScanActive { ExternalAccessible := 'False'; ExternalVisible := 'False'; ExternalWritable := 'False'} : Bool;   //  Acknowledgement of the no-scan mode. Open: The X-ray is not in the no-scan mode. Closed: The X-ray is in the no-scan mode.
      ix_ReadyToScan { ExternalAccessible := 'False'; ExternalVisible := 'False'; ExternalWritable := 'False'} : Bool;   //  Contract from XCT (Gantry Control) Closed: Gantry is ready and have the nominal Speed.
      ix_GINinMainTrack { ExternalAccessible := 'False'; ExternalVisible := 'False'; ExternalWritable := 'False'} : Bool;   //  GIN is detected in the tracking configured area
      ix_ResetEnergySave { ExternalAccessible := 'False'; ExternalVisible := 'False'; ExternalWritable := 'False'} : Bool;   //  Reset energy save mode timer
      ix_TakeoutConveyorRunning { ExternalAccessible := 'False'; ExternalVisible := 'False'; ExternalWritable := 'False'} : Bool;   //  Outfeef conveyor running
      ix_IQTestSelection { ExternalAccessible := 'False'; ExternalVisible := 'False'; ExternalWritable := 'False'} : Bool;   //  IQ test enable
      ix_IQTestStopPEC { ExternalAccessible := 'False'; ExternalVisible := 'False'; ExternalWritable := 'False'} : Bool;   //  IQ test outfeed conveyor stop PEC
   END_VAR

   VAR_OUTPUT
      qUDT_HMIStatus { ExternalAccessible := 'False'; ExternalVisible := 'False'; ExternalWritable := 'False'} : "UDT_HS10080XCTStatus";   //  HMI status structure
      qUDT_Status { ExternalAccessible := 'False'; ExternalVisible := 'False'; ExternalWritable := 'False'} : "UDT_CommonStatus";   //  Common status structure
      qx_NoScan { ExternalAccessible := 'False'; ExternalVisible := 'False'; ExternalWritable := 'False'} : Bool;   //  Request for the no-scan mode. Open: X-ray out of no-scan mode (screening mode). Closed: X-ray in no-scan mode.
      qx_InfeedConveyorOn { ExternalAccessible := 'False'; ExternalVisible := 'False'; ExternalWritable := 'False'} : Bool;   //  The infeed conveyor control. (HDX only in no-scan mode) Open: The BHS-PLC has no need for running the X-ray infeed conveyor. Closed: Run the X-ray infeed conveyor.
      qx_MainConveyorOn { ExternalAccessible := 'False'; ExternalVisible := 'False'; ExternalWritable := 'False'} : Bool;   //  The main conveyor control. (HDX only in no-scan mode) Open: The BHS-PLC has no need for running the X-ray main conveyor. Closed: Run the X-ray main conveyor.
      qx_OutfeedConveyorOn { ExternalAccessible := 'False'; ExternalVisible := 'False'; ExternalWritable := 'False'} : Bool;   //  The outfeed conveyor control. (HDX only in no-scan mode) Open: The BHS-PLC has no need for running the X-ray outfeed conveyor. Closed: Run the X-ray outfeed conveyor.
      qx_ESReset { ExternalAccessible := 'False'; ExternalVisible := 'False'; ExternalWritable := 'False'} : Bool;   //  Emergency stop reset. Open: No action. Closed: Resets the last emergency stop event. Must be closed for approximately 0.5 seconds.
      qx_PowerOn { ExternalAccessible := 'False'; ExternalVisible := 'False'; ExternalWritable := 'False'} : Bool;   //  Remote power-on for the X-ray. Open: Power down. Closed: Power up and start of initialisation.
      qx_PrepareToScan { ExternalAccessible := 'False'; ExternalVisible := 'False'; ExternalWritable := 'False'} : Bool;   //  Control of gantry rotation Closed: Gantry start rotation, acceleration time ~90 sec. Open: Gantry stop,decelerationtime ~100 sec,
      qx_ReadyForCal { ExternalAccessible := 'False'; ExternalVisible := 'False'; ExternalWritable := 'False'} : Bool;   //  Accept of Calibration request. Closed: External infeed conveyors are stopped. Waiting for calibration to end.
      qx_IQTestInfeedHold { ExternalAccessible := 'False'; ExternalVisible := 'False'; ExternalWritable := 'False'} : Bool;   //  IQ test infeed belt hold
      qx_IQTestOutfeedHold { ExternalAccessible := 'False'; ExternalVisible := 'False'; ExternalWritable := 'False'} : Bool;   //  IQ test outfeed belt hold
      qx_IQTestIndication { ExternalAccessible := 'False'; ExternalVisible := 'False'; ExternalWritable := 'False'} : Bool;   //  IQ test lamp indication
   END_VAR

   VAR_IN_OUT
      iqUDT_Statistics : "UDT_HS10080XCTStatistics";   //  Statistics structure
      iqUDT_EquipmentControl : "UDT_EquipmentControl";   //  Equipment control stucture
      iqUDT_InfeedConveyorInterface : "UDT_ConveyorInterface";   //  Infeed conveyor interface structure
      iqUDT_MainConveyorInterface : "UDT_ConveyorInterface";   //  Main conveyor interface structure
      iqUDT_OutfeedConveyorInterface : "UDT_ConveyorInterface";   //  Outfeed conveyor interface structure
      iqUDT_HandShakeUp : "UDT_ConveyorHandshake";   //  Upstream handshake structure
      iqUDT_Handshake : "UDT_ConveyorHandshake";   //  Downstream handshake structure
   END_VAR

   VAR
      sUDT_HMIStatus { ExternalAccessible := 'False'; ExternalVisible := 'False'; ExternalWritable := 'False'; S7_SetPoint := 'False'} : "UDT_HS10080XCTStatus";   //  HMI status structure
      sUDT_CommonStatusOld { ExternalAccessible := 'False'; ExternalVisible := 'False'; ExternalWritable := 'False'; S7_SetPoint := 'False'} : "UDT_CommonStatus";   //  Common status structure
      sUDT_CommonStatus { ExternalAccessible := 'False'; ExternalVisible := 'False'; ExternalWritable := 'False'; S7_SetPoint := 'False'} : "UDT_CommonStatus";   //  Common status structure
      sUDT_InfeedConvCommonStatus { ExternalAccessible := 'False'; ExternalVisible := 'False'; ExternalWritable := 'False'; S7_SetPoint := 'False'} : "UDT_CommonStatus";   //  Common status for infeed conveyor
      sUDT_MainConvCommonStatus { ExternalAccessible := 'False'; ExternalVisible := 'False'; ExternalWritable := 'False'; S7_SetPoint := 'False'} : "UDT_CommonStatus";   //  Common status for main conveyor
      sUDT_OutfeedConvCommonStatus { ExternalAccessible := 'False'; ExternalVisible := 'False'; ExternalWritable := 'False'; S7_SetPoint := 'False'} : "UDT_CommonStatus";   //  Common status for outfeed conveyor
      sUDT_InfeedConvCommonStatusOld { ExternalAccessible := 'False'; ExternalVisible := 'False'; ExternalWritable := 'False'; S7_SetPoint := 'False'} : "UDT_CommonStatus";   //  Common status for infeed conveyor
      sUDT_MainConvCommonStatusOld { ExternalAccessible := 'False'; ExternalVisible := 'False'; ExternalWritable := 'False'; S7_SetPoint := 'False'} : "UDT_CommonStatus";   //  Common status for main conveyor
      sUDT_OutfeedConvCommonStatusOld { ExternalAccessible := 'False'; ExternalVisible := 'False'; ExternalWritable := 'False'; S7_SetPoint := 'False'} : "UDT_CommonStatus";   //  Common status for outfeed conveyor
      s_OutfeedPECEoSFiltered { ExternalAccessible := 'False'; ExternalVisible := 'False'; ExternalWritable := 'False'; S7_SetPoint := 'False'} : "FB_TimerOnOffDelay";   //  Filtering end of section photo eye signal
      s_InfeedPECEoSFiltered { ExternalAccessible := 'False'; ExternalVisible := 'False'; ExternalWritable := 'False'; S7_SetPoint := 'False'} : "FB_TimerOnOffDelay";   //  Filtering end of section photo eye signal
      s_CascadeModeTimer { ExternalAccessible := 'False'; ExternalVisible := 'False'; ExternalWritable := 'False'; S7_SetPoint := 'False'} : "FB_TimerOnOffDelay";   //  Timer to cascade start
      s_CallibrationForceDelay { ExternalAccessible := 'False'; ExternalVisible := 'False'; ExternalWritable := 'False'; S7_SetPoint := 'False'} : "FB_TimerOnOffDelay";   //  Delay before callibration is forced on
      s_MainConvRunFeedback { ExternalAccessible := 'False'; ExternalVisible := 'False'; ExternalWritable := 'False'; S7_SetPoint := 'False'} : "FB_TimerOnOffDelay";   //  Conveyor run feeback
      s_IQTestRealese { ExternalAccessible := 'False'; ExternalVisible := 'False'; ExternalWritable := 'False'; S7_SetPoint := 'False'} : "FB_TimerOnOffDelay";   //  Conveyor run feeback
      s_EntryEncoderFault { ExternalAccessible := 'False'; ExternalVisible := 'False'; ExternalWritable := 'False'; S7_SetPoint := 'False'} : "FB_TimerOnOffDelay";   //  Entry encoder fault
      s_MainEncoderFault { ExternalAccessible := 'False'; ExternalVisible := 'False'; ExternalWritable := 'False'; S7_SetPoint := 'False'} : "FB_TimerOnOffDelay";   //  Main encoder fault
      s_ExitEncoderFault { ExternalAccessible := 'False'; ExternalVisible := 'False'; ExternalWritable := 'False'; S7_SetPoint := 'False'} : "FB_TimerOnOffDelay";   //  Exit encoder fault
      R_TRIG_Stop {InstructionName := 'R_TRIG'; LibVersion := '1.0'; ExternalAccessible := 'False'; ExternalVisible := 'False'; ExternalWritable := 'False'; S7_SetPoint := 'False'} : R_TRIG;   //  Rising edge trigger to stop conveyor
      R_TRIG_Running {InstructionName := 'R_TRIG'; LibVersion := '1.0'; ExternalAccessible := 'False'; ExternalVisible := 'False'; ExternalWritable := 'False'; S7_SetPoint := 'False'} : R_TRIG;   //  Rising edge trigger running
      R_TRIG_MainRunning {InstructionName := 'R_TRIG'; LibVersion := '1.0'; ExternalAccessible := 'False'; ExternalVisible := 'False'; ExternalWritable := 'False'; S7_SetPoint := 'False'} : R_TRIG;   //  Rising edge trigger running
      R_TRIG_OutfeedRunning {InstructionName := 'R_TRIG'; LibVersion := '1.0'; ExternalAccessible := 'False'; ExternalVisible := 'False'; ExternalWritable := 'False'; S7_SetPoint := 'False'} : R_TRIG;   //  Rising edge trigger running
      R_TRIG_XRayMode {InstructionName := 'R_TRIG'; LibVersion := '1.0'; ExternalAccessible := 'False'; ExternalVisible := 'False'; ExternalWritable := 'False'; S7_SetPoint := 'False'} : R_TRIG;   //  Rising edge trigger in X-ray mode
      R_TRIG_ServiceMode {InstructionName := 'R_TRIG'; LibVersion := '1.0'; ExternalAccessible := 'False'; ExternalVisible := 'False'; ExternalWritable := 'False'; S7_SetPoint := 'False'} : R_TRIG;   //  Rising edge trigger in service mode
      R_TRIG_TransitMode {InstructionName := 'R_TRIG'; LibVersion := '1.0'; ExternalAccessible := 'False'; ExternalVisible := 'False'; ExternalWritable := 'False'; S7_SetPoint := 'False'} : R_TRIG;   //  Rising edge trigger in transitmode
      R_TRIG_Estop {InstructionName := 'R_TRIG'; LibVersion := '1.0'; ExternalAccessible := 'False'; ExternalVisible := 'False'; ExternalWritable := 'False'; S7_SetPoint := 'False'} : R_TRIG;   //  Rising edge trigger E-stop active
      R_TRIG_RepairSwitch {InstructionName := 'R_TRIG'; LibVersion := '1.0'; ExternalAccessible := 'False'; ExternalVisible := 'False'; ExternalWritable := 'False'; S7_SetPoint := 'False'} : R_TRIG;   //  Rising edge trigger Repairswitch
      R_TRIG_TempOutOfRange {InstructionName := 'R_TRIG'; LibVersion := '1.0'; ExternalAccessible := 'False'; ExternalVisible := 'False'; ExternalWritable := 'False'; S7_SetPoint := 'False'} : R_TRIG;   //  Rising edge trigger Temperature Out Of Range
      R_TRIG_TailToBegin {InstructionName := 'R_TRIG'; LibVersion := '1.0'; ExternalAccessible := 'False'; ExternalVisible := 'False'; ExternalWritable := 'False'; S7_SetPoint := 'False'} : R_TRIG;   //  Rising edge trigger Tail arrive at the beginning of next conveyor
      R_TRIG_Calibrating {InstructionName := 'R_TRIG'; LibVersion := '1.0'; ExternalAccessible := 'False'; ExternalVisible := 'False'; ExternalWritable := 'False'; S7_SetPoint := 'False'} : R_TRIG;   //  Rising edge trigger Calibrating
      R_TRIG_CalibrationForce {InstructionName := 'R_TRIG'; LibVersion := '1.0'; ExternalAccessible := 'False'; ExternalVisible := 'False'; ExternalWritable := 'False'; S7_SetPoint := 'False'} : R_TRIG;   //  Rising edge trigger Callibration is forced
      R_TRIG_InfConvErr {InstructionName := 'R_TRIG'; LibVersion := '1.0'; ExternalAccessible := 'False'; ExternalVisible := 'False'; ExternalWritable := 'False'; S7_SetPoint := 'False'} : R_TRIG;   //  Rising edge trigger Infeed conveyor error
      R_TRIG_OutfConvErr {InstructionName := 'R_TRIG'; LibVersion := '1.0'; ExternalAccessible := 'False'; ExternalVisible := 'False'; ExternalWritable := 'False'; S7_SetPoint := 'False'} : R_TRIG;   //  Rising edge trigger Outfeed conveyor error
      R_TRIG_EncoderErr {InstructionName := 'R_TRIG'; LibVersion := '1.0'; ExternalAccessible := 'False'; ExternalVisible := 'False'; ExternalWritable := 'False'; S7_SetPoint := 'False'} : R_TRIG;   //  Rising edge trigger encoder error
      F_TRIG_Callibrating {InstructionName := 'F_TRIG'; LibVersion := '1.0'; ExternalAccessible := 'False'; ExternalVisible := 'False'; ExternalWritable := 'False'; S7_SetPoint := 'False'} : F_TRIG;   //  Falling edge trigger Callibrating
      F_TRIG_Interlock {InstructionName := 'F_TRIG'; LibVersion := '1.0'; ExternalAccessible := 'False'; ExternalVisible := 'False'; ExternalWritable := 'False'; S7_SetPoint := 'False'} : F_TRIG;   //  Falling edge trigger Interlock
      R_TRIG_PEC_EoSFiltered {InstructionName := 'R_TRIG'; LibVersion := '1.0'; ExternalAccessible := 'False'; ExternalVisible := 'False'; ExternalWritable := 'False'; S7_SetPoint := 'False'} : R_TRIG;   //  Rising edge trigger end of section photo eye filtered
      F_TRIG_PEC_EosFiltered {InstructionName := 'F_TRIG'; LibVersion := '1.0'; ExternalAccessible := 'False'; ExternalVisible := 'False'; ExternalWritable := 'False'; S7_SetPoint := 'False'} : F_TRIG;   //  Falling edge PEC EOS
      F_TRIG_SignalingRequest {InstructionName := 'F_TRIG'; LibVersion := '1.0'; ExternalAccessible := 'False'; ExternalVisible := 'False'; ExternalWritable := 'False'; S7_SetPoint := 'False'} : F_TRIG;   //  Falling edge signaling request
      F_TRIG_EnergySaveActive {InstructionName := 'F_TRIG'; LibVersion := '1.0'; ExternalAccessible := 'False'; ExternalVisible := 'False'; ExternalWritable := 'False'; S7_SetPoint := 'False'} : F_TRIG;   //  Falling edge Energy save active
      F_TRIG_AuxHeadToEnd {InstructionName := 'F_TRIG'; LibVersion := '1.0'; ExternalAccessible := 'False'; ExternalVisible := 'False'; ExternalWritable := 'False'; S7_SetPoint := 'False'} : F_TRIG;   //  Falling edge trigger Aux head to end bit
      R_TRIG_TakeoutConveyorRuning {InstructionName := 'R_TRIG'; LibVersion := '1.0'; ExternalAccessible := 'False'; ExternalVisible := 'False'; ExternalWritable := 'False'; S7_SetPoint := 'False'} : R_TRIG;   //  Falling edge trigger takeout conveyors running
      R_TRIG_IQTest {InstructionName := 'R_TRIG'; LibVersion := '1.0'; ExternalAccessible := 'False'; ExternalVisible := 'False'; ExternalWritable := 'False'; S7_SetPoint := 'False'} : R_TRIG;   //  Falling edge trigger takeout conveyors running
   END_VAR
   VAR RETAIN
      sdi_DistanceStopping { ExternalAccessible := 'False'; ExternalVisible := 'False'; ExternalWritable := 'False'} : DInt;   //  Actual distance after stop signal (cm)
   END_VAR
   VAR
      sdi_PECOutfeedDistanceOffset { ExternalAccessible := 'False'; ExternalVisible := 'False'; ExternalWritable := 'False'} : DInt;   //  Distance offset between photo eye and the end of conveyor [mm]
   END_VAR
   VAR RETAIN
      sdi_DistanceRunEmptyMain { ExternalAccessible := 'False'; ExternalVisible := 'False'; ExternalWritable := 'False'} : DInt;   //  Actual distance running empty
      sdi_DistanceRunEmptyOutfeed { ExternalAccessible := 'False'; ExternalVisible := 'False'; ExternalWritable := 'False'} : DInt;   //  Actual distance running empty
   END_VAR
   VAR
      sdi_ClearDistance { ExternalAccessible := 'False'; ExternalVisible := 'False'; ExternalWritable := 'False'} : DInt;   //  Distance on takeout conveyor to clear before start
      si_IQTestEmptyDistance { ExternalAccessible := 'False'; ExternalVisible := 'False'; ExternalWritable := 'False'} : Int;
   END_VAR
   VAR RETAIN
      si_GapTailToHead { ExternalAccessible := 'False'; ExternalVisible := 'False'; ExternalWritable := 'False'} : Int;   //  Actual size gap tail to head
      si_OutfeedAuxJamDisplacement { ExternalAccessible := 'False'; ExternalVisible := 'False'; ExternalWritable := 'False'} : Int;   //  Auxiliary variable to calculate displacement when PEC is blocked
      si_InfeedAuxJamDisplacement { ExternalAccessible := 'False'; ExternalVisible := 'False'; ExternalWritable := 'False'} : Int;   //  Auxiliary variable to calculate displacement when PEC is blocked
      si_AuxEnergySave { ExternalAccessible := 'False'; ExternalVisible := 'False'; ExternalWritable := 'False'} : Int;   //  Auxiliary variable to calculate energy save displacement
      si_TailToBegin { ExternalAccessible := 'False'; ExternalVisible := 'False'; ExternalWritable := 'False'} : Int;   //  Count tail to next conveyor distance
      si_HeadToEnd { ExternalAccessible := 'False'; ExternalVisible := 'False'; ExternalWritable := 'False'} : Int;   //  Count head to end distance
      sx_AuxHeadToEnd { ExternalAccessible := 'False'; ExternalVisible := 'False'; ExternalWritable := 'False'} : Bool;   //  Aux bit to control head to end positioning
      sx_AuxHeadAtEnd { ExternalAccessible := 'False'; ExternalVisible := 'False'; ExternalWritable := 'False'} : Bool;   //  Aux bit to memorise head at end positioning
      sx_TailToBegin { ExternalAccessible := 'False'; ExternalVisible := 'False'; ExternalWritable := 'False'} : Bool;   //  Trail to begin done
      sx_EnergySaveActive { ExternalAccessible := 'False'; ExternalVisible := 'False'; ExternalWritable := 'False'} : Bool;   //  Active energy save mode
   END_VAR
   VAR
      sx_PEC_OutfeedEoSFiltered { ExternalAccessible := 'False'; ExternalVisible := 'False'; ExternalWritable := 'False'} : Bool;   //  End of section photo eye filtered
      sx_PEC_InfeedEoSFiltered { ExternalAccessible := 'False'; ExternalVisible := 'False'; ExternalWritable := 'False'} : Bool;   //  End of section photo eye filtered
      sx_MainConvReady { ExternalAccessible := 'False'; ExternalVisible := 'False'; ExternalWritable := 'False'} : Bool;   //  Conveyor Ready to operate in Automatic mode
      sx_StartReceived { ExternalAccessible := 'False'; ExternalVisible := 'False'; ExternalWritable := 'False'} : Bool;   //  Start command received from system
      sx_MainAutomaticActive { ExternalAccessible := 'False'; ExternalVisible := 'False'; ExternalWritable := 'False'} : Bool;   //  Running in automatic
      sx_OutfeedAutomaticActive { ExternalAccessible := 'False'; ExternalVisible := 'False'; ExternalWritable := 'False'} : Bool;   //  Running in automatic
      sx_ManualModeActive { ExternalAccessible := 'False'; ExternalVisible := 'False'; ExternalWritable := 'False'} : Bool;   //  Manual mode active
      sx_RunningEmptyMain { ExternalAccessible := 'False'; ExternalVisible := 'False'; ExternalWritable := 'False'} : Bool;   //  X-Ray main is running empty
      sx_RunningEmptyOutfeed { ExternalAccessible := 'False'; ExternalVisible := 'False'; ExternalWritable := 'False'} : Bool;   //  X-Ray outfeed is running empty
      sx_ReqToCal { ExternalAccessible := 'False'; ExternalVisible := 'False'; ExternalWritable := 'False'} : Bool;   //  Request to calibrate received
      sx_ParcelAtEnd { ExternalAccessible := 'False'; ExternalVisible := 'False'; ExternalWritable := 'False'} : Bool;   //  Parcel is detected in window at end of main conveyor
      sx_Stopping { ExternalAccessible := 'False'; ExternalVisible := 'False'; ExternalWritable := 'False'} : Bool;   //  Stopping seuence is activated
      sx_Stopped { ExternalAccessible := 'False'; ExternalVisible := 'False'; ExternalWritable := 'False'} : Bool;   //  Stopping sequence is ended
      sx_Gapping { ExternalAccessible := 'False'; ExternalVisible := 'False'; ExternalWritable := 'False'} : Bool;   //  The outfeed conveyor is creating a gap downstream
      sx_calibrating { ExternalAccessible := 'False'; ExternalVisible := 'False'; ExternalWritable := 'False'} : Bool;   //  XCT Calibration is ongoing
      sx_CallibrateForceOn { ExternalAccessible := 'False'; ExternalVisible := 'False'; ExternalWritable := 'False'} : Bool;   //  XCT Callibration is forced on because wating timed out
      sx_MainConvRunFeedbackError { ExternalAccessible := 'False'; ExternalVisible := 'False'; ExternalWritable := 'False'} : Bool;   //  Main conveyor running feedback error
      sx_MachineHealthy { ExternalAccessible := 'False'; ExternalVisible := 'False'; ExternalWritable := 'False'} : Bool;   //  Machine healthy status
      sx_ResetRunEmptyESave { ExternalAccessible := 'False'; ExternalVisible := 'False'; ExternalWritable := 'False'} : Bool;   //  Resent energy save to run empty
      sx_MainConveyorOn { ExternalAccessible := 'False'; ExternalVisible := 'False'; ExternalWritable := 'False'} : Bool;   //  Main conveyor control
      sx_ReadyForCal { ExternalAccessible := 'False'; ExternalVisible := 'False'; ExternalWritable := 'False'} : Bool;   //  Ready for calibration
      sx_TakeoutConveyorClear { ExternalAccessible := 'False'; ExternalVisible := 'False'; ExternalWritable := 'False'} : Bool;   //  Takeout conveyor clear
      sx_IQTestReady { ExternalAccessible := 'False'; ExternalVisible := 'False'; ExternalWritable := 'False'} : Bool;
      sx_InfeedConveyorOn { ExternalAccessible := 'False'; ExternalVisible := 'False'; ExternalWritable := 'False'} : Bool;   //  Infeed conveyor control
      sx_OutfeedConveyorOn { ExternalAccessible := 'False'; ExternalVisible := 'False'; ExternalWritable := 'False'} : Bool;   //  Oufeed conveyor control
   END_VAR

   VAR_TEMP
      tx_PowerOn : Bool;   //  Startup the machine
      tx_PrepareToScan : Bool;   //  Power on X-Ray generator
   END_VAR


BEGIN
	(*
	----------------------------------------------------------------------------------------

	Version history:
	Date        | Version   | Author        | Remark
	----------------------------------------------------------------------------------------
	29/05/2019  | 0.1       | Frank Baten   | first release TIA 15
	24/07/2019  | 2.0       | L.Klar        | 2.0 MHS library release TIA 15.1
	07/08/2019  | 2.1       | S.Theocharis  | 2.1 Updates during test at SMITHS Detection
	09/08/2019  | 2.2       | Frank Baten   | 2.2 Add control of infeed conveyor
	13/08/2019  | 2.3       | S.Theocharis  | 2.3 Updated with interface of infeed conveyor
	20/08/2019  | 2.4       | S.Theocharis  | 2.4 Add the internal tracking error
	26/08/2019  | 2.5       | S.Theocharis  | Update the "UDT_HS10080XCT_Configuration"
	25/09/2019  | 2.6       | S. Deulkar    | Created 3 different entity for 3 conveyor, automatic active, error etc.
	                                        | Added infeed PEC blockage logic
	                                        | Modified logic for Infeed and outfeed conveyor run
	                                        | Adeed 3 status and report block call for 3 xray belts
	                                        | No scan HMI command is added,ON commands output activates
	11/10/2019  | 2.7       | S.Deulkar     | Update new status structure
	04/11/2019  | 2.8       | L.Klar        | First scan bit changed from memory bit to DB variable
	12/11/2019  | 3.0       | P.Majka       | 3.0 MHS library release TIA 15.1
	13/01/2020  | 3.2       | F.Baten       | Changed length related tags from Int to Dint
	11/01/2021  | 3.3       | L.Klar        | Sinput safety ok added to stop conveyor condition
	09/02/2021  | 3.4       | L.Klar        | IQ test added
	04/03/2021  | 3.5       | M.Kurpiers    | HMI status updated - xray ready warning added
	13/03/2021  | 3.6       | L.Klar        | HMI status updated- warning commented, energy save added, diaback added when machine in startup
	20/03/2021  | 3.7       | L.Klar        | Encoders errors added
	09/06/2021  | 3.8       | M.Kurpiers    | E-Stop Active statistics changed
	04/04/2023  | 4.0       | F.Baten       | 4.0 Release TIA 17.5
	*)

	REGION 1 - Initial and Calibration

	    // First PLC cycle
	    IF "DB_Memory".FirstScan
	    THEN
	        #sx_MainAutomaticActive := FALSE;                                                                           // switch of automatic activ
	        #iqUDT_HandShakeUp.RTR := False;                                                                           // Reset RTR signal
	        #iqUDT_HandShakeUp.CascadeStartUp := FALSE;                                                                // Reset cascade start signal
	        #sx_Stopping := FALSE;                                                                                      // Reset stopping sequence
	        #sx_Stopped := TRUE;                                                                                        // Set machine is stopped
	    END_IF;

	    // Calibrating Condition
	    (* Xray do not share calibrating status with PLC, hence follwoing condtions are used to check if machine is calibrating)*)
	    #sx_calibrating := #ix_CalReq AND #sx_ReadyForCal AND NOT #ix_XrayReady;

	END_REGION

	REGION 2 - Triggers
	    // Statement section REGION

	    #R_TRIG_XRayMode(CLK := NOT #sUDT_CommonStatus.Stopped AND NOT #ix_ServiceMode AND NOT #ix_TransitActive);      // Rising edge trigger X-Ray mode

	    #R_TRIG_ServiceMode(CLK := NOT #sUDT_CommonStatus.Stopped AND #ix_ServiceMode);                                 // Rising edge trigger in service mode

	    #R_TRIG_TransitMode(CLK := NOT #sUDT_CommonStatus.Stopped AND #ix_TransitActive);                               // Rising edge trigger in transitmode

	    #R_TRIG_Estop(CLK := NOT #ix_SafetyOk);                                                                          // Rising edge trigger E-stop active

	    #R_TRIG_RepairSwitch(CLK := #ix_RepairSwitch);                                                                   // Rising edge trigger Repairswitch

	    #R_TRIG_TempOutOfRange(CLK := #ix_TempOutOfRange);                                                               // Rising edge trigger Temperature Out Of Range

	    #R_TRIG_Calibrating(CLK := #sx_calibrating);                                                                     // Rising edge trigger Calibrating

	    #F_TRIG_Interlock(CLK := #ix_Interlock);                                                                         // Falling edge trigger interlock (1=ok)

	    #R_TRIG_Running(CLK := #sUDT_CommonStatus.Running);                                                             // Rising edge trigger running X-Ray system

	    #R_TRIG_Stop(CLK := #sUDT_CommonStatus.Stopped);                                                                // Rising edge trigger x-ray stopped

	    #R_TRIG_MainRunning(CLK := #ix_MainSpeedOk);                                                                     // Rising edge trigger running main conveyor

	    #F_TRIG_Callibrating(CLK := #sx_calibrating);                                                                    // Falling edge trigger callibrating

	    #R_TRIG_PEC_EoSFiltered(CLK := #sx_PEC_OutfeedEoSFiltered);                                                      // Rising edge trigger PEC EOS

	    #F_TRIG_PEC_EosFiltered(CLK := #sx_PEC_OutfeedEoSFiltered);                                                      // Falling edge trigger PEC EOS

	    #F_TRIG_SignalingRequest(CLK := #iqUDT_EquipmentControl.Request.SignalingRequest); // Falling edge trigger signaling request

	    #R_TRIG_TakeoutConveyorRuning(CLK := #ix_TakeoutConveyorRunning);


	    // PEC Filter
	    #s_OutfeedPECEoSFiltered(iudi_OnDelayTime := #iUDT_EquipmentConfiguration.PEC_OutfeedTimeOnDelay,
	                             iudi_OffDelayTime := #iUDT_EquipmentConfiguration.PEC_OutfeedTimeOffDelay,
	                             ix_SignalToDelay := #ix_PECOutfeedEoS,
	                             ix_Enable := TRUE,
	                             qx_DelayedSignal => #sx_PEC_OutfeedEoSFiltered);

	    #s_InfeedPECEoSFiltered(iudi_OnDelayTime := #iUDT_EquipmentConfiguration.PEC_InfeedTimeOnDelay,
	                            iudi_OffDelayTime := #iUDT_EquipmentConfiguration.PEC_InfeedTimeOffDelay,
	                            ix_SignalToDelay := #ix_PECInfeedEoS,
	                            ix_Enable := TRUE,
	                            qx_DelayedSignal => #sx_PEC_InfeedEoSFiltered);

	END_REGION

	REGION 3 - Error handling
	    REGION 3.1 - Reset Errors
	        IF #iqUDT_EquipmentControl.Command.Reset                                                                   // If Reset command appeared from system control
	        THEN

	            IF #sUDT_HMIStatus.OutfeedConvSpecific.PEC_EoSJam                                                          // If Outfeed EOS PEC Jammed error is active
	                AND ((#iUDT_EquipmentConfiguration.ResetWithPECBlocked)                                            // And Reset with PEC blocked is enabled
	                OR (NOT #iUDT_EquipmentConfiguration.ResetWithPECBlocked AND #sx_PEC_OutfeedEoSFiltered))          // Or reset is not enabled and PEC is unblocked
	            THEN                                                                                                    // Then
	                #sUDT_HMIStatus.OutfeedConvSpecific.PEC_EoSJam := FALSE;                                               // reset PEC jam error
	            END_IF;

	            IF #sUDT_HMIStatus.InfeedConvSpecific.PEC_EoSJam                                                           // If Infeed EOS PEC Jammed error is active
	                AND ((#iUDT_EquipmentConfiguration.ResetWithPECBlocked)                                            // And Reset with PEC blocked is enabled
	                OR (NOT #iUDT_EquipmentConfiguration.ResetWithPECBlocked AND #sx_PEC_InfeedEoSFiltered))           // Or reset is not enabled and PEC is unblocked
	            THEN                                                                                                    // Then
	                #sUDT_HMIStatus.InfeedConvSpecific.PEC_EoSJam := FALSE;                                                // reset PEC jam error
	            END_IF;
	            #sx_MainConvRunFeedbackError := FALSE;
	            #sUDT_HMIStatus.InfeedConvSpecific.Conv_ERR := FALSE;                                                      // Reset infeed conveyor feedback error
	            #sUDT_HMIStatus.MainConvSpecific.Conv_ERR := FALSE;                                                        // Reset main conveyor feedback error
	            #sUDT_HMIStatus.OutfeedConvSpecific.Conv_ERR := FALSE;
	            #sUDT_HMIStatus.InfeedConvSpecific.Encoder_ERR := FALSE;                                                      // Reset infeed conveyor feedback error
	            #sUDT_HMIStatus.MainConvSpecific.Encoder_ERR := FALSE;                                                        // Reset main conveyor feedback error
	            #sUDT_HMIStatus.OutfeedConvSpecific.Encoder_ERR := FALSE;     // Reset outfeed conveyor feedback error
	        END_IF;
	    END_REGION

	    REGION 3.2 - Xray Errors
	        // Xray machine errors / Warnings
	        #sUDT_HMIStatus.XraySpecific.DoorInterlockNotOk := NOT #ix_Interlock;                                 // One of the doors of the in or outfeed tunnel is opend
	        #sUDT_HMIStatus.XraySpecific.RepairSwitch := #ix_RepairSwitch;                                        // X-ray mains are powered off
	        #sUDT_HMIStatus.XraySpecific.ServiceMode := #ix_ServiceMode;                                          // The X-ray is in service mode.
	        #sUDT_HMIStatus.XraySpecific.TempOutOfRange := #ix_TempOutOfRange;                                    // XCT doesn’t work because XCT operating temperature isn’t given
	        #sUDT_HMIStatus.XraySpecific.GantrySpeedNotOk := NOT #ix_ReadyToScan;                                 // Gantry speed is not Ok
	        #sUDT_HMIStatus.XraySpecific.IQTestActive := #ix_IQTestSelection OR #ix_IQTestActive;                                        // IQ test is active on XRAY
	        #sUDT_HMIStatus.XraySpecific.XrayPowerNotOn := NOT #ix_PowerOn;                                       // Power is not switched on
	        #sUDT_HMIStatus.XraySpecific.MachineNotOk := NOT #ix_MachineOk;                                       // Machine is not ok
	        #sUDT_HMIStatus.XraySpecific.XRayNotReady := NOT #ix_XrayReady;                                       // X-Ray is not ready to operate
	        #sUDT_HMIStatus.XraySpecific.TransitActive := #ix_TransitActive;                                      // The transit mode is active
	        #sUDT_HMIStatus.XraySpecific.NoScanActive := #ix_NoScanActive;                                        // The X-ray is in the no-scan mode.

	        // Xray Common "Error"
	        #sUDT_CommonStatus.Error := NOT #ix_24vOk                                                                  // 24v signalling not OK
	        OR NOT #ix_400vOk                                                                                           // 400v signalling not OK
	        OR NOT #ix_ProfinetOk                                                                                       // Profinet signalling not OK
	        OR NOT #ix_SafetyOk
	        OR #sUDT_HMIStatus.XraySpecific.MachineNotOk                                                                                         // Safety signalling NOT OK
	        // changed onsite
	        OR NOT #sUDT_HMIStatus.XraySpecific.RepairSwitch                                                                   // X-ray mains are powered off
	        OR #sUDT_InfeedConvCommonStatus.Error                                                                          // Or error is active on main conveyor
	        OR #sUDT_MainConvCommonStatus.Error                                                                            // Or error is active on main conveyor
	        OR #sUDT_OutfeedConvCommonStatus.Error
	        OR (#sUDT_HMIStatus.XraySpecific.ServiceMode AND NOT #ix_IQTestSelection)                                                                    // The X-ray is in service mode.
	        OR #sUDT_HMIStatus.XraySpecific.TempOutOfRange;                                                                // XCT doesn’t work because XCT operating temperature isn’t given
	        //OR #s_StatusUDT.XraySpecific.GantrySpeedNotOk                                                             // Xraay gantry speed is not ok

	    END_REGION

	    REGION 3.3 - Infeed conveyor errors

	        IF #ix_InfConveyorError OR #iqUDT_InfeedConveyorInterface.InternalErrorTracking THEN                                                                        // If main conveyor feedback error active then
	            #sUDT_HMIStatus.InfeedConvSpecific.Conv_ERR := TRUE;                                                       // Create infeed conveyor feedback error
	        END_IF;

	        #s_EntryEncoderFault(iudi_OnDelayTime := 5000,
	                             ix_SignalToDelay := #sx_InfeedConveyorOn AND #iqUDT_InfeedConveyorInterface.Displacement = 0,                         //If Main conveyor speed not Ok
	                             ix_Enable := TRUE);

	        IF #s_EntryEncoderFault.qx_DelayedSignal THEN
	            #sUDT_HMIStatus.InfeedConvSpecific.Encoder_ERR := TRUE;
	        END_IF;

	        IF NOT #sx_PEC_InfeedEoSFiltered                                                                            // PEC is blocked
	        THEN
	            #si_InfeedAuxJamDisplacement += #iqUDT_InfeedConveyorInterface.Displacement;                          // Increase memory with actual displacement
	        ELSE
	            #si_InfeedAuxJamDisplacement := 0;                                                                     // Reset memory (PEC was free)
	        END_IF;

	        IF #si_InfeedAuxJamDisplacement > #iUDT_EquipmentConfiguration.InfeedPECJamDisplacementLimit THEN         // If memory is bigger than setpoint, set error
	            #sUDT_HMIStatus.InfeedConvSpecific.PEC_EoSJam := TRUE;
	        END_IF;

	        #sUDT_InfeedConvCommonStatus.Error := #sUDT_HMIStatus.InfeedConvSpecific.PEC_EoSJam                               // Infeed conveyor PEC Jammed
	        OR #sUDT_HMIStatus.InfeedConvSpecific.Conv_ERR                                                                 // Infeed conveyor is in error
	        OR #sUDT_HMIStatus.InfeedConvSpecific.Encoder_ERR;                                                             // Infeed conveyor has encoder error

	    END_REGION

	    REGION 3.4 - Main conveyor Errors

	        #s_MainEncoderFault(iudi_OnDelayTime := 5000,
	                            ix_SignalToDelay := #sx_MainConveyorOn AND #ix_MainSpeedOk AND #iqUDT_MainConveyorInterface.Displacement = 0,                         //If Main conveyor speed not Ok
	                            ix_Enable := TRUE);

	        IF #s_MainEncoderFault.qx_DelayedSignal THEN
	            #sUDT_HMIStatus.MainConvSpecific.Encoder_ERR := TRUE;
	        END_IF;                                            // The Main conveyor encoder is faulted

	        #s_MainConvRunFeedback(iudi_OnDelayTime := #iUDT_EquipmentConfiguration.MainConvFeedbackDelayTime,
	                               ix_SignalToDelay := #sx_MainConveyorOn AND NOT #ix_MainSpeedOk,                         //If Main conveyor speed not Ok
	                               ix_Enable := TRUE,                                                                       // Enable timer when run command to main conveyor is ON
	                               qx_DelayedSignal => #sx_MainConvRunFeedbackError);

	        IF #sx_MainConvRunFeedbackError OR #iqUDT_MainConveyorInterface.InternalErrorTracking THEN                                                                        // If main conveyor feedback error active then
	            #sUDT_HMIStatus.MainConvSpecific.Conv_ERR := TRUE;                                                         // Create main conveyor feedback error
	        END_IF;

	        #sUDT_MainConvCommonStatus.Error :=
	        #sUDT_HMIStatus.MainConvSpecific.Conv_ERR                                                                      // Outfeed conveyor is in error
	        OR #sUDT_HMIStatus.MainConvSpecific.Encoder_ERR;

	    END_REGION

	    REGION 3.5 - Outfeed conveyor errors

	        IF #ix_OutfConveyorError OR #iqUDT_OutfeedConveyorInterface.InternalErrorTracking THEN                                                                        // If main conveyor feedback error active then
	            #sUDT_HMIStatus.OutfeedConvSpecific.Conv_ERR := TRUE;                                                      // Create infeed conveyor feedback error
	        END_IF;

	        #s_ExitEncoderFault(iudi_OnDelayTime := 5000,
	                            ix_SignalToDelay := #sx_OutfeedConveyorOn AND #iqUDT_OutfeedConveyorInterface.Displacement = 0,                         //If Main conveyor speed not Ok
	                            ix_Enable := TRUE);

	        IF #s_ExitEncoderFault.qx_DelayedSignal THEN
	            #sUDT_HMIStatus.OutfeedConvSpecific.Encoder_ERR := TRUE;
	        END_IF;                                       // The Infeed conveyor encoder is faulted

	        IF NOT #sx_PEC_OutfeedEoSFiltered                                                                           // PEC is blocked
	        THEN
	            #si_OutfeedAuxJamDisplacement += #iqUDT_OutfeedConveyorInterface.Displacement;                        // Increase memory with actual displacement
	        ELSE
	            #si_OutfeedAuxJamDisplacement := 0;                                                                    // Reset memory (PEC was free)
	        END_IF;

	        IF #si_OutfeedAuxJamDisplacement > #iUDT_EquipmentConfiguration.OutfeedPECJamDisplacementLimit THEN       // If memory is bigger than setpoint, set error
	            #sUDT_HMIStatus.OutfeedConvSpecific.PEC_EoSJam := TRUE;
	        END_IF;

	        #sUDT_OutfeedConvCommonStatus.Error := #sUDT_HMIStatus.OutfeedConvSpecific.PEC_EoSJam                             // Outfeed conveyor PEC Jammed
	        OR #sUDT_HMIStatus.OutfeedConvSpecific.Conv_ERR                                                                // Outfeed conveyor is in error
	        OR #sUDT_HMIStatus.OutfeedConvSpecific.Encoder_ERR;                                                            // Outfeed conveyor has encoder error
	    END_REGION

	    // Common warning
	    #sUDT_CommonStatus.Warning :=
	    #sUDT_HMIStatus.XraySpecific.TransitActive                                                                         // The transit mode is active
	    OR #sUDT_HMIStatus.XraySpecific.NoScanActive                                                                      // The X-ray is in the no-scan mode.
	    OR #sUDT_HMIStatus.XraySpecific.DoorInterlockNotOk // Interlock open
	    OR #sUDT_HMIStatus.XraySpecific.XRayNotReady;
	    //Conditions to set bit sx_Ready to operate
	    #sx_MainConvReady := NOT #sUDT_CommonStatus.Error AND NOT #sUDT_MainConvCommonStatus.Error;

	END_REGION

	REGION 4 - Stop Equipment
	    (* When a stop command is received the machine will transport the parcels to the end of the machine
	       so clearing the main conveyor. If the main conveyor is stopped (because of a parcel in the last position)
	       or the main conveyor has run its emptying distance the machine will stop.*)

	    IF NOT #iqUDT_EquipmentControl.Command.AutomaticOn                                                             // if Stop active from system control ( Means Not automatic ON)
	        AND NOT #iqUDT_EquipmentControl.Command.Start                                                              // And no start command from system control
	        AND #sx_MainAutomaticActive                                                                                 // And system is Automatic active
	    THEN                                                                                                            // Then
	        IF NOT #sx_Stopping THEN                                                                                    // If Stopping sequence is not activated
	            #sdi_DistanceStopping := 0; //((#i_UDT_EquipmentConfiguration.InfeedConveyor.Length +
	            // #i_UDT_EquipmentConfiguration.MainConveyor.Length +
	            // #i_UDT_EquipmentConfiguration.OutfeedConveyor.Length + 1000) / 10);                                            // Calculate stopping distance in cm
	        END_IF;
	        #sx_Stopping := TRUE;                                                                                       // Activate stop sequence
	    END_IF;

	    IF #sx_Stopping THEN                                                                                            // If stopping sequence is activated then
	        #sdi_DistanceStopping -= #iqUDT_MainConveyorInterface.Displacement;                                         // Calculate stopping distance

	        IF #sdi_DistanceStopping < 0                                                                                 // And if stopping distance is done
	            OR NOT #ix_MainSpeedOk                                                                                  // or if main conveyor is not already stopped
	        THEN                                                                                                        // Then
	            #sx_Stopped := TRUE;                                                                                    // make Stopped status TRUE
	            #sx_Stopping := FALSE;                                                                                  // and Reset stopping sequence
	        END_IF;
	    END_IF;

	    //Main and outfeed conveyor
	    IF #sx_Stopped                                                                                                  // If Stop command received and both conveyors are stopped
	        OR #sUDT_CommonStatus.Error                                                                                // Or an error is active on Xray Or error is active on main conveyor
	        OR (#ix_TransitActive AND NOT #sx_IQTestReady)                                                                                   // AND Xray is not in transit mode
	        //OR (#ix_ServiceMode AND NOT #ix_IQTestSelection)                                                                                          // AND Xray is not in service mode
	        OR NOT #ix_SafetyOk
	        //OR (#i_UDT_HMICommand.NoScanMode AND NOT #ix_ReadyToScan)
	    THEN                                                                                                            // Then
	        #iqUDT_HandShakeUp.RTR := FALSE;                                                                           // Reset RTR signal
	        #iqUDT_HandShakeUp.CascadeStartUp := FALSE;                                                                // Reset cascade start signal
	        #sx_MainAutomaticActive := FALSE;                                                                           // Switch off automatic active
	        #sx_OutfeedAutomaticActive := FALSE;                                                                        // Switch off automatic active
	        #sx_StartReceived := FALSE;                                                                                 // Reset start command received from system
	    END_IF;

	END_REGION

	REGION 5 - Start Automatic mode
	    // if start (OS) is received from system, this is memorised until started in cascade
	    IF #iqUDT_EquipmentControl.Command.Start                                                                       // If Start command from from system received

	    THEN                                                                                                            // Then
	        #sx_StartReceived := TRUE;                                                                                  // Set Start command received from system
	        #sx_Stopping := FALSE;                                                                                      // Stop stopping sequence
	        #sx_Stopped := FALSE;                                                                                       // Reset stopped bit
	    END_IF;

	    IF #sx_StartReceived                                                                                            // If Start command received from system
	        AND (#iqUDT_Handshake.CascadeStartUp                                                                       // Handshake from downstream conveyor to cascade start
	        OR #iUDT_EquipmentConfiguration.FirstConveyorToStart)                                                      // of if this is the first conveyor to start in the cascade
	    THEN                                                                                                            // THEN
	        #sx_MainAutomaticActive := TRUE;                                                                            // Set Automatic active
	        #sx_OutfeedAutomaticActive := TRUE;                                                                         // Set Automatic active
	        #sx_StartReceived := FALSE;                                                                                 // and reset start received bit
	    END_IF;

	    // Cascade mode
	    #s_CascadeModeTimer(iudi_OnDelayTime := #iUDT_EquipmentConfiguration.CascadeTimeOnDelay,                       //Timer to cascade mode--Outfeed Conveyor
	                        ix_SignalToDelay := #sx_MainAutomaticActive,
	                        ix_Enable := #sUDT_InfeedConvCommonStatus.Running,
	                        qx_DelayedSignal => #iqUDT_HandShakeUp.CascadeStartUp);

	    #sx_ManualModeActive := FALSE;                                                                                  // No manual mode available for Xray machine hence disabled it.
	END_REGION

	REGION 6 - Automatic mode active
	    REGION 6.1 - Head to End
	        (*  Function to calculate when the head of the parcel reaches the end of the conveyor
	            When the PEC detects the parcels head, the functionality increments the displacement
	            of the conveyor until it reaches the value of the distance between PEC and the end of the conveyor.
	            After that, the counter is reset and the bit #sx_AuxHeadToEnd is triggered to inform the system. *)
	        #sdi_PECOutfeedDistanceOffset := #iUDT_EquipmentConfiguration.PEC_OutfeedDistanceOffset;

	        IF #sdi_PECOutfeedDistanceOffset >= #iUDT_EquipmentConfiguration.PEC_OutfeedDistance
	        THEN
	            #sdi_PECOutfeedDistanceOffset := #iUDT_EquipmentConfiguration.PEC_OutfeedDistance - 1;
	        END_IF;

	        IF #F_TRIG_PEC_EosFiltered.Q THEN                                                                           // If the product's head is detected then
	            #si_HeadToEnd := (#iUDT_EquipmentConfiguration.PEC_OutfeedDistance                                     // Move PEC distand minus PEC offset to static variable in cm
	            - #iUDT_EquipmentConfiguration.PEC_OutfeedDistanceOffset) / 10;                                        // (Static variable is virtual distance between PEC and end of the conveyor)

	            #sx_AuxHeadToEnd := TRUE;                                                                               //And active head to end function
	            #iqUDT_Handshake.RTS := TRUE;                                                                          //And Set Ready TO Send true when a parcel is detected in the PEC
	        END_IF;

